LIN {X 0,Y 298.466,Z 479.305,A -85,B 0,C 180,E1 -16236.813,E2 -16236.813} C_VEL
LIN {X 0,Y 298.452,Z 479.311,A -85,B 0,C 180,E1 -16241.25,E2 -16241.25} C_VEL
LIN {X 0,Y 298.537,Z 479.479,A -85,B 0,C 180,E1 -16243.984,E2 -16243.984} C_VEL
LIN {X 0,Y 299.451,Z 484.848,A -85,B 0,C 180,E1 -16247.917,E2 -16247.917} C_VEL
LIN {X 0,Y 300.419,Z 490.228,A -85,B 0,C 180,E1 -16251.688,E2 -16251.688} C_VEL
LIN {X 0,Y 300.571,Z 494.055,A -85,B 0,C 180,E1 -16254.229,E2 -16254.229} C_VEL
LIN {X 0,Y 299.738,Z 499.296,A -85,B 0,C 180,E1 -16257.575,E2 -16257.575} C_VEL
LIN {X 0,Y 298.893,Z 505.042,A -85,B 0,C 180,E1 -16261.182,E2 -16261.182} C_VEL
LIN {X 0,Y 297.961,Z 512.224,A -85,B 0,C 180,E1 -16265.621,E2 -16265.621} C_VEL
LIN {X 0,Y 297.495,Z 517.191,A -85,B 0,C 180,E1 -16268.634,E2 -16268.634} C_VEL
LIN {X 0,Y 298.743,Z 530.872,A -85,B 0,C 180,E1 -16269.444,E2 -16269.444} C_VEL
LIN {X 0,Y 300.095,Z 544.162,A -85,B 0,C 180,E1 -16270.512,E2 -16270.512} C_VEL
LIN {X 0,Y 301.357,Z 557.073,A -85,B 0,C 180,E1 -16271.825,E2 -16271.825} C_VEL
LIN {X 0,Y 301.113,Z 562.88,A -85,B 0,C 180,E1 -16272.512,E2 -16272.512} C_VEL
LIN {X 0,Y 299.918,Z 574.212,A -85,B 0,C 180,E1 -16274.077,E2 -16274.077} C_VEL
LIN {X 0,Y 298.966,Z 583.854,A -85,B 0,C 180,E1 -16275.71,E2 -16275.71} C_VEL
LIN {X 0,Y 298.052,Z 593.552,A -85,B 0,C 180,E1 -16277.748,E2 -16277.748} C_VEL
LIN {X 0,Y 297.384,Z 601.387,A -85,B 0,C 180,E1 -16279.791,E2 -16279.791} C_VEL
LIN {X 0,Y 297.034,Z 607.671,A -85,B 0,C 180,E1 -16281.839,E2 -16281.839} C_VEL
LIN {X 0,Y 296.864,Z 612.635,A -85,B 0,C 180,E1 -16283.887,E2 -16283.887} C_VEL
LIN {X 0,Y 296.808,Z 616.412,A -85,B 0,C 180,E1 -16285.927,E2 -16285.927} C_VEL
LIN {X 0,Y 296.812,Z 618.317,A -85,B 0,C 180,E1 -16287.286,E2 -16287.286} C_VEL
LIN {X 0,Y 296.996,Z 619.803,A -85,B 0,C 180,E1 -16288.644,E2 -16288.644} C_VEL
LIN {X 0,Y 296.994,Z 620.81,A -85,B 0,C 180,E1 -16290,E2 -16290} C_VEL
LIN {X 0,Y 296.862,Z 621.357,A -85,B 0,C 180,E1 -16291.357,E2 -16291.357} C_VEL
LIN {X 0,Y 296.64,Z 621.229,A -85,B 0,C 180,E1 -16294.076,E2 -16294.076} C_VEL
LIN {X 0,Y 296.595,Z 620.43,A -85,B 0,C 180,E1 -16295.607,E2 -16295.607} C_VEL
LIN {X 0,Y 296.89,Z 617.954,A -85,B 0,C 180,E1 -16298.166,E2 -16298.166} C_VEL
LIN {X 0,Y 297.683,Z 613.764,A -85,B 0,C 180,E1 -16300.887,E2 -16300.887} C_VEL
LIN {X 0,Y 298.649,Z 609.478,A -85,B 0,C 180,E1 -16302.919,E2 -16302.919} C_VEL
LIN {X 0,Y 300.437,Z 603.094,A -85,B 0,C 180,E1 -16305.258,E2 -16305.258} C_VEL
LIN {X 0,Y 302.414,Z 595.236,A -85,B 0,C 180,E1 -16307.585,E2 -16307.585} C_VEL
LIN {X 0,Y 304.966,Z 586.959,A -85,B 0,C 180,E1 -16309.522,E2 -16309.522} C_VEL
LIN {X 0,Y 307.811,Z 577.052,A -85,B 0,C 180,E1 -16311.427,E2 -16311.427} C_VEL
LIN {X 0,Y 309.967,Z 569.372,A -85,B 0,C 180,E1 -16312.672,E2 -16312.672} C_VEL
LIN {X 0,Y 311.299,Z 559.086,A -85,B 0,C 180,E1 -16314.278,E2 -16314.278} C_VEL
LIN {X 0,Y 311.377,Z 550.475,A -85,B 0,C 180,E1 -16315.638,E2 -16315.638} C_VEL
LIN {X 0,Y 310.206,Z 538.996,A -85,B 0,C 180,E1 -16317.496,E2 -16317.496} C_VEL
LIN {X 0,Y 307.841,Z 527.667,A -85,B 0,C 180,E1 -16319.496,E2 -16319.496} C_VEL
LIN {X 0,Y 305.431,Z 518.991,A -85,B 0,C 180,E1 -16321.194,E2 -16321.194} C_VEL
LIN {X 0,Y 303.143,Z 512.4,A -85,B 0,C 180,E1 -16322.676,E2 -16322.676} C_VEL
LIN {X 0,Y 301.622,Z 508.711,A -85,B 0,C 180,E1 -16323.642,E2 -16323.642} C_VEL
LIN {X 0,Y 301.271,Z 506.687,A -85,B 0,C 180,E1 -16324.047,E2 -16324.047} C_VEL
LIN {X 0,Y 302.094,Z 503.342,A -85,B 0,C 180,E1 -16327.22,E2 -16327.22} C_VEL
LIN {X 0,Y 302.148,Z 501.053,A -85,B 0,C 180,E1 -16329.863,E2 -16329.863} C_VEL
LIN {X 0,Y 301.802,Z 498.422,A -85,B 0,C 180,E1 -16333.789,E2 -16333.789} C_VEL
LIN {X 0,Y 301.46,Z 496.683,A -85,B 0,C 180,E1 -16337.462,E2 -16337.462} C_VEL
LIN {X 0,Y 301.194,Z 495.638,A -85,B 0,C 180,E1 -16340.949,E2 -16340.949} C_VEL
LIN {X 0,Y 300.84,Z 495.191,A -85,B 0,C 180,E1 -16344.266,E2 -16344.266} C_VEL
LIN {X 0,Y 300.63,Z 495.276,A -85,B 0,C 180,E1 -16345.923,E2 -16345.923} C_VEL
LIN {X 0,Y 301.106,Z 496.736,A -85,B 0,C 180,E1 -16346.358,E2 -16346.358} C_VEL
LIN {X 0,Y 301.952,Z 498.177,A -85,B 0,C 180,E1 -16346.921,E2 -16346.921} C_VEL
LIN {X 0,Y 303.759,Z 499.965,A -85,B 0,C 180,E1 -16347.85,E2 -16347.85} C_VEL
LIN {X 0,Y 304.765,Z 502.419,A -85,B 0,C 180,E1 -16348.566,E2 -16348.566} C_VEL
LIN {X 0,Y 306.416,Z 504.69,A -85,B 0,C 180,E1 -16349.405,E2 -16349.405} C_VEL
LIN {X 0,Y 306.908,Z 506.071,A -85,B 0,C 180,E1 -16349.749,E2 -16349.749} C_VEL
LIN {X 0,Y 308.354,Z 508.316,A -85,B 0,C 180,E1 -16350.508,E2 -16350.508} C_VEL
LIN {X 0,Y 312.476,Z 517.896,A -85,B 0,C 180,E1 -16352.944,E2 -16352.944} C_VEL
LIN {X 0,Y 315.184,Z 526.862,A -85,B 0,C 180,E1 -16354.934,E2 -16354.934} C_VEL
LIN {X 0,Y 316.223,Z 532.587,A -85,B 0,C 180,E1 -16356.098,E2 -16356.098} C_VEL
LIN {X 0,Y 312.862,Z 544.975,A -85,B 0,C 180,E1 -16357.898,E2 -16357.898} C_VEL
LIN {X 0,Y 309.781,Z 555.156,A -85,B 0,C 180,E1 -16359.759,E2 -16359.759} C_VEL
LIN {X 0,Y 306.983,Z 563.531,A -85,B 0,C 180,E1 -16361.652,E2 -16361.652} C_VEL
LIN {X 0,Y 304.706,Z 570.437,A -85,B 0,C 180,E1 -16363.588,E2 -16363.588} C_VEL
LIN {X 0,Y 302.42,Z 576.841,A -85,B 0,C 180,E1 -16365.877,E2 -16365.877} C_VEL
LIN {X 0,Y 300.729,Z 581.193,A -85,B 0,C 180,E1 -16367.859,E2 -16367.859} C_VEL
LIN {X 0,Y 299.962,Z 583.522,A -85,B 0,C 180,E1 -16369.197,E2 -16369.197} C_VEL
LIN {X 0,Y 299.12,Z 585.612,A -85,B 0,C 180,E1 -16370.687,E2 -16370.687} C_VEL
LIN {X 0,Y 297.885,Z 588.001,A -85,B 0,C 180,E1 -16373.226,E2 -16373.226} C_VEL
LIN {X 0,Y 297.69,Z 588.691,A -85,B 0,C 180,E1 -16374.582,E2 -16374.582} C_VEL
LIN {X 0,Y 297.438,Z 589,A -85,B 0,C 180,E1 -16375.935,E2 -16375.935} C_VEL
LIN {X 0,Y 296.934,Z 588.398,A -85,B 0,C 180,E1 -16378.644,E2 -16378.644} C_VEL
LIN {X 0,Y 296.812,Z 587.512,A -85,B 0,C 180,E1 -16380,E2 -16380} C_VEL
LIN {X 0,Y 296.762,Z 586.21,A -85,B 0,C 180,E1 -16381.357,E2 -16381.357} C_VEL
LIN {X 0,Y 296.845,Z 583.461,A -85,B 0,C 180,E1 -16383.394,E2 -16383.394} C_VEL
LIN {X 0,Y 297.012,Z 579.68,A -85,B 0,C 180,E1 -16385.432,E2 -16385.432} C_VEL
LIN {X 0,Y 297.346,Z 574.78,A -85,B 0,C 180,E1 -16387.47,E2 -16387.47} C_VEL
LIN {X 0,Y 297.88,Z 567.471,A -85,B 0,C 180,E1 -16389.849,E2 -16389.849} C_VEL
LIN {X 0,Y 298.614,Z 559.653,A -85,B 0,C 180,E1 -16391.885,E2 -16391.885} C_VEL
LIN {X 0,Y 299.575,Z 549.967,A -85,B 0,C 180,E1 -16393.914,E2 -16393.914} C_VEL
LIN {X 0,Y 300.544,Z 540.158,A -85,B 0,C 180,E1 -16395.6,E2 -16395.6} C_VEL
LIN {X 0,Y 301.436,Z 530.908,A -85,B 0,C 180,E1 -16396.92,E2 -16396.92} C_VEL
LIN {X 0,Y 302.482,Z 519.263,A -85,B 0,C 180,E1 -16398.281,E2 -16398.281} C_VEL
LIN {X 0,Y 302.839,Z 514.221,A -85,B 0,C 180,E1 -16398.784,E2 -16398.784} C_VEL
LIN {X 0,Y 300.737,Z 502.562,A -85,B 0,C 180,E1 -16399.877,E2 -16399.877} C_VEL
LIN {X 0,Y 298.12,Z 489.054,A -85,B 0,C 180,E1 -16400.877,E2 -16400.877} C_VEL
LIN {X 0,Y 297.077,Z 483.361,A -85,B 0,C 180,E1 -16401.239,E2 -16401.239} C_VEL
LIN {X 0,Y 297.196,Z 479.837,A -85,B 0,C 180,E1 -16405.193,E2 -16405.193} C_VEL
LIN {X 0,Y 297.331,Z 479.45,A -85,B 0,C 180,E1 -16406.687,E2 -16406.687} C_VEL
LIN {X 0,Y 297.686,Z 479.402,A -85,B 0,C 180,E1 -16409.722,E2 -16409.722} C_VEL
LIN {X 0,Y 297.986,Z 479.364,A -85,B 0,C 180,E1 -16412.852,E2 -16412.852} C_VEL
LIN {X 0,Y 298.373,Z 479.317,A -85,B 0,C 180,E1 -16416.788,E2 -16416.788} C_VEL
LIN {X 0,Y 298.399,Z 479.312,A -85,B 0,C 180,E1 -16419.488,E2 -16419.488} C_VEL
LIN {X 0,Y 298.402,Z 479.311,A -85,B 0,C 180,E1 -16423.103,E2 -16423.103} C_VEL
LIN {X 0,Y 298.407,Z 479.312,A -85,B 0,C 180,E1 -16426.921,E2 -16426.921} C_VEL
LIN {X 0,Y 298.419,Z 479.309,A -85,B 0,C 180,E1 -16431.004,E2 -16431.004} C_VEL
LIN {X 0,Y 298.425,Z 479.312,A -85,B 0,C 180,E1 -16433.931,E2 -16433.931} C_VEL
LIN {X 0,Y 298.399,Z 479.316,A -85,B 0,C 180,E1 -16437.984,E2 -16437.984} C_VEL
LIN {X 0,Y 298.463,Z 479.307,A -85,B 0,C 180,E1 -16441.904,E2 -16441.904} C_VEL
LIN {X 0,Y 298.49,Z 479.301,A -85,B 0,C 180,E1 -16444.924,E2 -16444.924} C_VEL
LIN {X 0,Y 298.455,Z 479.305,A -85,B 0,C 180,E1 -16449.315,E2 -16449.315} C_VEL
LIN {X 0,Y 298.543,Z 479.299,A -85,B 0,C 180,E1 -16452.179,E2 -16452.179} C_VEL
LIN {X 0,Y 298.598,Z 479.287,A -85,B 0,C 180,E1 -16454.995,E2 -16454.995} C_VEL
LIN {X 0,Y 298.597,Z 479.287,A -85,B 0,C 180,E1 -16459.146,E2 -16459.146} C_VEL
LIN {X 0,Y 298.745,Z 479.273,A -85,B 0,C 180,E1 -16461.885,E2 -16461.885} C_VEL
LIN {X 0,Y 298.661,Z 479.28,A -85,B 0,C 180,E1 -16464.599,E2 -16464.599} C_VEL
LIN {X 0,Y 298.927,Z 479.247,A -85,B 0,C 180,E1 -16468.653,E2 -16468.653} C_VEL
LIN {X 0,Y 298.929,Z 479.247,A -85,B 0,C 180,E1 -16471.347,E2 -16471.347} C_VEL
LIN {X 0,Y 298.649,Z 479.281,A -85,B 0,C 180,E1 -16475.401,E2 -16475.401} C_VEL
LIN {X 0,Y 298.718,Z 479.276,A -85,B 0,C 180,E1 -16478.115,E2 -16478.115} C_VEL
LIN {X 0,Y 298.558,Z 479.294,A -85,B 0,C 180,E1 -16482.231,E2 -16482.231} C_VEL
LIN {X 0,Y 298.61,Z 479.286,A -85,B 0,C 180,E1 -16485.209,E2 -16485.209} C_VEL
LIN {X 0,Y 298.544,Z 479.295,A -85,B 0,C 180,E1 -16489.243,E2 -16489.243} C_VEL
LIN {X 0,Y 298.461,Z 479.307,A -85,B 0,C 180,E1 -16493.597,E2 -16493.597} C_VEL
LIN {X 0,Y 298.49,Z 479.301,A -85,B 0,C 180,E1 -16496.574,E2 -16496.574} C_VEL
LIN {X 0,Y 298.419,Z 479.313,A -85,B 0,C 180,E1 -16499.641,E2 -16499.641} C_VEL
LIN {X 0,Y 298.398,Z 479.312,A -85,B 0,C 180,E1 -16502.8,E2 -16502.8} C_VEL
LIN {X 0,Y 298.467,Z 479.303,A -85,B 0,C 180,E1 -16506.812,E2 -16506.812} C_VEL
LIN {X 0,Y 298.389,Z 479.313,A -85,B 0,C 180,E1 -16511.087,E2 -16511.087} C_VEL
LIN {X 0,Y 298.4,Z 479.313,A -85,B 0,C 180,E1 -16513.103,E2 -16513.103} C_VEL
LIN {X 0,Y 298.404,Z 479.311,A -85,B 0,C 180,E1 -16516.92,E2 -16516.92} C_VEL
LIN {X 0,Y 298.416,Z 479.31,A -85,B 0,C 180,E1 -16521.003,E2 -16521.003} C_VEL
LIN {X 0,Y 298.42,Z 479.313,A -85,B 0,C 180,E1 -16523.93,E2 -16523.93} C_VEL
LIN {X 0,Y 298.397,Z 479.315,A -85,B 0,C 180,E1 -16527.983,E2 -16527.983} C_VEL
LIN {X 0,Y 298.465,Z 479.307,A -85,B 0,C 180,E1 -16531.904,E2 -16531.904} C_VEL
LIN {X 0,Y 298.487,Z 479.301,A -85,B 0,C 180,E1 -16534.924,E2 -16534.924} C_VEL
LIN {X 0,Y 298.451,Z 479.308,A -85,B 0,C 180,E1 -16539.315,E2 -16539.315} C_VEL
LIN {X 0,Y 298.539,Z 479.295,A -85,B 0,C 180,E1 -16542.179,E2 -16542.179} C_VEL
LIN {X 0,Y 298.594,Z 479.288,A -85,B 0,C 180,E1 -16544.994,E2 -16544.994} C_VEL
LIN {X 0,Y 298.595,Z 479.29,A -85,B 0,C 180,E1 -16549.146,E2 -16549.146} C_VEL
LIN {X 0,Y 298.759,Z 479.269,A -85,B 0,C 180,E1 -16551.886,E2 -16551.886} C_VEL
LIN {X 0,Y 298.661,Z 479.279,A -85,B 0,C 180,E1 -16554.599,E2 -16554.599} C_VEL
LIN {X 0,Y 298.925,Z 479.247,A -85,B 0,C 180,E1 -16558.652,E2 -16558.652} C_VEL
LIN {X 0,Y 298.924,Z 479.25,A -85,B 0,C 180,E1 -16561.347,E2 -16561.347} C_VEL
LIN {X 0,Y 298.618,Z 479.284,A -85,B 0,C 180,E1 -16563.886,E2 -16563.886} C_VEL
LIN {X 0,Y 297.887,Z 479.382,A -85,B 0,C 180,E1 -16565.012,E2 -16565.012} C_VEL
LIN {X 0,Y 295.114,Z 479.733,A -85,B 0,C 180,E1 -16566.85,E2 -16566.85} C_VEL
LIN {X 0,Y 291.972,Z 480.118,A -85,B 0,C 180,E1 -16569.104,E2 -16569.104} C_VEL
LIN {X 0,Y 291.609,Z 480.159,A -85,B 0,C 180,E1 -16569.881,E2 -16569.881} C_VEL
LIN {X 0,Y 291.522,Z 480.17,A -85,B 0,C 180,E1 -16573.95,E2 -16573.95} C_VEL
LIN {X 0,Y 291.487,Z 480.174,A -85,B 0,C 180,E1 -16576.818,E2 -16576.818} C_VEL
LIN {X 0,Y 291.45,Z 480.178,A -85,B 0,C 180,E1 -16579.875,E2 -16579.875} C_VEL
LIN {X 0,Y 291.399,Z 480.184,A -85,B 0,C 180,E1 -16584.205,E2 -16584.205} C_VEL
LIN {X 0,Y 291.418,Z 480.186,A -85,B 0,C 180,E1 -16587.272,E2 -16587.272} C_VEL
LIN {X 0,Y 291.334,Z 480.192,A -85,B 0,C 180,E1 -16590.437,E2 -16590.437} C_VEL
LIN {X 0,Y 291.344,Z 480.193,A -85,B 0,C 180,E1 -16593.698,E2 -16593.698} C_VEL
LIN {X 0,Y 291.399,Z 480.188,A -85,B 0,C 180,E1 -16597.26,E2 -16597.26} C_VEL
LIN {X 0,Y 291.4,Z 480.185,A -85,B 0,C 180,E1 -16600.631,E2 -16600.631} C_VEL
LIN {X 0,Y 291.489,Z 480.238,A -85,B 0,C 180,E1 -16603.748,E2 -16603.748} C_VEL
LIN {X 0,Y 292.493,Z 486.094,A -85,B 0,C 180,E1 -16608.147,E2 -16608.147} C_VEL
LIN {X 0,Y 293.31,Z 490.731,A -85,B 0,C 180,E1 -16611.466,E2 -16611.466} C_VEL
LIN {X 0,Y 293.549,Z 493.289,A -85,B 0,C 180,E1 -16613.235,E2 -16613.235} C_VEL
LIN {X 0,Y 293.16,Z 497.014,A -85,B 0,C 180,E1 -16615.711,E2 -16615.711} C_VEL
LIN {X 0,Y 292.082,Z 503.661,A -85,B 0,C 180,E1 -16620.023,E2 -16620.023} C_VEL
LIN {X 0,Y 291.131,Z 510.266,A -85,B 0,C 180,E1 -16624.245,E2 -16624.245} C_VEL
LIN {X 0,Y 290.418,Z 517.025,A -85,B 0,C 180,E1 -16628.39,E2 -16628.39} C_VEL
LIN {X 0,Y 291.665,Z 530.669,A -85,B 0,C 180,E1 -16629.225,E2 -16629.225} C_VEL
LIN {X 0,Y 293.019,Z 544.552,A -85,B 0,C 180,E1 -16630.38,E2 -16630.38} C_VEL
LIN {X 0,Y 294.281,Z 557.344,A -85,B 0,C 180,E1 -16631.733,E2 -16631.733} C_VEL
LIN {X 0,Y 293.898,Z 564.374,A -85,B 0,C 180,E1 -16632.608,E2 -16632.608} C_VEL
LIN {X 0,Y 292.718,Z 575.145,A -85,B 0,C 180,E1 -16634.181,E2 -16634.181} C_VEL
LIN {X 0,Y 291.697,Z 585.479,A -85,B 0,C 180,E1 -16636.059,E2 -16636.059} C_VEL
LIN {X 0,Y 290.819,Z 594.796,A -85,B 0,C 180,E1 -16638.147,E2 -16638.147} C_VEL
LIN {X 0,Y 290.249,Z 602.267,A -85,B 0,C 180,E1 -16640.242,E2 -16640.242} C_VEL
LIN {X 0,Y 289.929,Z 608.278,A -85,B 0,C 180,E1 -16642.339,E2 -16642.339} C_VEL
LIN {X 0,Y 289.863,Z 613.015,A -85,B 0,C 180,E1 -16644.435,E2 -16644.435} C_VEL
LIN {X 0,Y 289.753,Z 615.522,A -85,B 0,C 180,E1 -16645.827,E2 -16645.827} C_VEL
LIN {X 0,Y 289.74,Z 617.505,A -85,B 0,C 180,E1 -16647.22,E2 -16647.22} C_VEL
LIN {X 0,Y 289.938,Z 619.053,A -85,B 0,C 180,E1 -16648.611,E2 -16648.611} C_VEL
LIN {X 0,Y 289.939,Z 620.147,A -85,B 0,C 180,E1 -16650,E2 -16650} C_VEL
LIN {X 0,Y 289.773,Z 620.789,A -85,B 0,C 180,E1 -16651.39,E2 -16651.39} C_VEL
LIN {X 0,Y 289.551,Z 620.801,A -85,B 0,C 180,E1 -16654.176,E2 -16654.176} C_VEL
LIN {X 0,Y 289.602,Z 619.229,A -85,B 0,C 180,E1 -16656.97,E2 -16656.97} C_VEL
LIN {X 0,Y 290.21,Z 616.025,A -85,B 0,C 180,E1 -16659.76,E2 -16659.76} C_VEL
LIN {X 0,Y 291.286,Z 611.2,A -85,B 0,C 180,E1 -16662.542,E2 -16662.542} C_VEL
LIN {X 0,Y 292.75,Z 606.428,A -85,B 0,C 180,E1 -16664.6,E2 -16664.6} C_VEL
LIN {X 0,Y 294.73,Z 599.496,A -85,B 0,C 180,E1 -16666.985,E2 -16666.985} C_VEL
LIN {X 0,Y 297.014,Z 592.228,A -85,B 0,C 180,E1 -16668.987,E2 -16668.987} C_VEL
LIN {X 0,Y 299.844,Z 583.583,A -85,B 0,C 180,E1 -16670.944,E2 -16670.944} C_VEL
LIN {X 0,Y 302.506,Z 575.043,A -85,B 0,C 180,E1 -16672.541,E2 -16672.541} C_VEL
LIN {X 0,Y 304.015,Z 569.384,A -85,B 0,C 180,E1 -16673.502,E2 -16673.502} C_VEL
LIN {X 0,Y 305.303,Z 561.033,A -85,B 0,C 180,E1 -16674.885,E2 -16674.885} C_VEL
LIN {X 0,Y 305.532,Z 551.878,A -85,B 0,C 180,E1 -16676.418,E2 -16676.418} C_VEL
LIN {X 0,Y 304.602,Z 541.064,A -85,B 0,C 180,E1 -16678.31,E2 -16678.31} C_VEL
LIN {X 0,Y 302.739,Z 531.064,A -85,B 0,C 180,E1 -16680.23,E2 -16680.23} C_VEL
LIN {X 0,Y 300.864,Z 523.19,A -85,B 0,C 180,E1 -16681.895,E2 -16681.895} C_VEL
LIN {X 0,Y 299.552,Z 518.592,A -85,B 0,C 180,E1 -16682.969,E2 -16682.969} C_VEL
LIN {X 0,Y 297.801,Z 513.56,A -85,B 0,C 180,E1 -16684.311,E2 -16684.311} C_VEL
LIN {X 0,Y 297.659,Z 512.608,A -85,B 0,C 180,E1 -16684.518,E2 -16684.518} C_VEL
LIN {X 0,Y 295.612,Z 508.107,A -85,B 0,C 180,E1 -16686.067,E2 -16686.067} C_VEL
LIN {X 0,Y 295.034,Z 505.141,A -85,B 0,C 180,E1 -16686.918,E2 -16686.918} C_VEL
LIN {X 0,Y 295.199,Z 503.926,A -85,B 0,C 180,E1 -16688.244,E2 -16688.244} C_VEL
LIN {X 0,Y 295.16,Z 502.235,A -85,B 0,C 180,E1 -16690.364,E2 -16690.364} C_VEL
LIN {X 0,Y 294.894,Z 500.053,A -85,B 0,C 180,E1 -16693.721,E2 -16693.721} C_VEL
LIN {X 0,Y 294.53,Z 498.2,A -85,B 0,C 180,E1 -16697.708,E2 -16697.708} C_VEL
LIN {X 0,Y 294.354,Z 497.513,A -85,B 0,C 180,E1 -16699.86,E2 -16699.86} C_VEL
LIN {X 0,Y 294.116,Z 497.014,A -85,B 0,C 180,E1 -16702.839,E2 -16702.839} C_VEL
LIN {X 0,Y 295.223,Z 499.509,A -85,B 0,C 180,E1 -16704.038,E2 -16704.038} C_VEL
LIN {X 0,Y 297.165,Z 501.335,A -85,B 0,C 180,E1 -16705.417,E2 -16705.417} C_VEL
LIN {X 0,Y 298.652,Z 504.229,A -85,B 0,C 180,E1 -16706.606,E2 -16706.606} C_VEL
LIN {X 0,Y 300.119,Z 505.816,A -85,B 0,C 180,E1 -16707.462,E2 -16707.462} C_VEL
LIN {X 0,Y 301.121,Z 508.24,A -85,B 0,C 180,E1 -16708.239,E2 -16708.239} C_VEL
LIN {X 0,Y 301.971,Z 509.364,A -85,B 0,C 180,E1 -16708.742,E2 -16708.742} C_VEL
LIN {X 0,Y 304.883,Z 515.521,A -85,B 0,C 180,E1 -16710.662,E2 -16710.662} C_VEL
LIN {X 0,Y 308.306,Z 524.86,A -85,B 0,C 180,E1 -16713.119,E2 -16713.119} C_VEL
LIN {X 0,Y 310.177,Z 532.971,A -85,B 0,C 180,E1 -16715.003,E2 -16715.003} C_VEL
LIN {X 0,Y 310.364,Z 534.297,A -85,B 0,C 180,E1 -16715.289,E2 -16715.289} C_VEL
LIN {X 0,Y 309.843,Z 537.437,A -85,B 0,C 180,E1 -16715.785,E2 -16715.785} C_VEL
LIN {X 0,Y 306.669,Z 547.839,A -85,B 0,C 180,E1 -16717.427,E2 -16717.427} C_VEL
LIN {X 0,Y 303.434,Z 557.555,A -85,B 0,C 180,E1 -16719.316,E2 -16719.316} C_VEL
LIN {X 0,Y 300.51,Z 565.566,A -85,B 0,C 180,E1 -16721.242,E2 -16721.242} C_VEL
LIN {X 0,Y 297.689,Z 573.08,A -85,B 0,C 180,E1 -16723.543,E2 -16723.543} C_VEL
LIN {X 0,Y 295.7,Z 578.283,A -85,B 0,C 180,E1 -16725.549,E2 -16725.549} C_VEL
LIN {X 0,Y 293.904,Z 582.416,A -85,B 0,C 180,E1 -16727.572,E2 -16727.572} C_VEL
LIN {X 0,Y 293.078,Z 584.589,A -85,B 0,C 180,E1 -16728.94,E2 -16728.94} C_VEL
LIN {X 0,Y 291.473,Z 587.758,A -85,B 0,C 180,E1 -16731.682,E2 -16731.682} C_VEL
LIN {X 0,Y 290.873,Z 588.76,A -85,B 0,C 180,E1 -16733.062,E2 -16733.062} C_VEL
LIN {X 0,Y 290.635,Z 589.327,A -85,B 0,C 180,E1 -16734.45,E2 -16734.45} C_VEL
LIN {X 0,Y 290.369,Z 589.505,A -85,B 0,C 180,E1 -16735.836,E2 -16735.836} C_VEL
LIN {X 0,Y 289.845,Z 588.74,A -85,B 0,C 180,E1 -16738.611,E2 -16738.611} C_VEL
LIN {X 0,Y 289.717,Z 587.746,A -85,B 0,C 180,E1 -16740,E2 -16740} C_VEL
LIN {X 0,Y 289.673,Z 586.323,A -85,B 0,C 180,E1 -16741.391,E2 -16741.391} C_VEL
LIN {X 0,Y 289.777,Z 583.417,A -85,B 0,C 180,E1 -16743.476,E2 -16743.476} C_VEL
LIN {X 0,Y 289.947,Z 578.622,A -85,B 0,C 180,E1 -16745.965,E2 -16745.965} C_VEL
LIN {X 0,Y 290.396,Z 572.51,A -85,B 0,C 180,E1 -16748.35,E2 -16748.35} C_VEL
LIN {X 0,Y 291.071,Z 564.428,A -85,B 0,C 180,E1 -16750.786,E2 -16750.786} C_VEL
LIN {X 0,Y 291.897,Z 555.777,A -85,B 0,C 180,E1 -16752.869,E2 -16752.869} C_VEL
LIN {X 0,Y 293.033,Z 545.097,A -85,B 0,C 180,E1 -16754.941,E2 -16754.941} C_VEL
LIN {X 0,Y 294.202,Z 534.097,A -85,B 0,C 180,E1 -16756.659,E2 -16756.659} C_VEL
LIN {X 0,Y 295.258,Z 521.873,A -85,B 0,C 180,E1 -16758.205,E2 -16758.205} C_VEL
LIN {X 0,Y 295.753,Z 515.364,A -85,B 0,C 180,E1 -16758.892,E2 -16758.892} C_VEL
LIN {X 0,Y 294.403,Z 506.887,A -85,B 0,C 180,E1 -16759.734,E2 -16759.734} C_VEL
LIN {X 0,Y 292.017,Z 494.407,A -85,B 0,C 180,E1 -16760.767,E2 -16760.767} C_VEL
LIN {X 0,Y 290.011,Z 483.742,A -85,B 0,C 180,E1 -16761.502,E2 -16761.502} C_VEL
LIN {X 0,Y 290.054,Z 481.255,A -85,B 0,C 180,E1 -16764.325,E2 -16764.325} C_VEL
LIN {X 0,Y 290.218,Z 480.336,A -85,B 0,C 180,E1 -16765.843,E2 -16765.843} C_VEL
LIN {X 0,Y 290.616,Z 480.282,A -85,B 0,C 180,E1 -16769.472,E2 -16769.472} C_VEL
LIN {X 0,Y 290.907,Z 480.25,A -85,B 0,C 180,E1 -16772.267,E2 -16772.267} C_VEL
LIN {X 0,Y 291.182,Z 480.211,A -85,B 0,C 180,E1 -16775.4,E2 -16775.4} C_VEL
LIN {X 0,Y 291.319,Z 480.194,A -85,B 0,C 180,E1 -16777.239,E2 -16777.239} C_VEL
LIN {X 0,Y 291.335,Z 480.193,A -85,B 0,C 180,E1 -16780.643,E2 -16780.643} C_VEL
LIN {X 0,Y 291.294,Z 480.201,A -85,B 0,C 180,E1 -16784.402,E2 -16784.402} C_VEL
LIN {X 0,Y 291.33,Z 480.196,A -85,B 0,C 180,E1 -16788.404,E2 -16788.404} C_VEL
LIN {X 0,Y 291.368,Z 480.187,A -85,B 0,C 180,E1 -16791.16,E2 -16791.16} C_VEL
LIN {X 0,Y 291.366,Z 480.19,A -85,B 0,C 180,E1 -16794.626,E2 -16794.626} C_VEL
LIN {X 0,Y 291.376,Z 480.19,A -85,B 0,C 180,E1 -16797.951,E2 -16797.951} C_VEL
LIN {X 0,Y 291.382,Z 480.186,A -85,B 0,C 180,E1 -16801.158,E2 -16801.158} C_VEL
LIN {X 0,Y 291.419,Z 480.186,A -85,B 0,C 180,E1 -16804.272,E2 -16804.272} C_VEL
LIN {X 0,Y 291.387,Z 480.185,A -85,B 0,C 180,E1 -16807.3,E2 -16807.3} C_VEL
LIN {X 0,Y 291.463,Z 480.18,A -85,B 0,C 180,E1 -16810.27,E2 -16810.27} C_VEL
LIN {X 0,Y 291.56,Z 480.165,A -85,B 0,C 180,E1 -16814.624,E2 -16814.624} C_VEL
LIN {X 0,Y 291.54,Z 480.166,A -85,B 0,C 180,E1 -16818.88,E2 -16818.88} C_VEL
LIN {X 0,Y 291.692,Z 480.15,A -85,B 0,C 180,E1 -16821.688,E2 -16821.688} C_VEL
LIN {X 0,Y 291.631,Z 480.156,A -85,B 0,C 180,E1 -16824.468,E2 -16824.468} C_VEL
LIN {X 0,Y 291.893,Z 480.123,A -85,B 0,C 180,E1 -16828.62,E2 -16828.62} C_VEL
LIN {X 0,Y 291.895,Z 480.123,A -85,B 0,C 180,E1 -16831.379,E2 -16831.379} C_VEL
LIN {X 0,Y 291.617,Z 480.158,A -85,B 0,C 180,E1 -16835.532,E2 -16835.532} C_VEL
LIN {X 0,Y 291.678,Z 480.149,A -85,B 0,C 180,E1 -16838.919,E2 -16838.919} C_VEL
LIN {X 0,Y 291.525,Z 480.168,A -85,B 0,C 180,E1 -16842.531,E2 -16842.531} C_VEL
LIN {X 0,Y 291.559,Z 480.165,A -85,B 0,C 180,E1 -16845.376,E2 -16845.376} C_VEL
LIN {X 0,Y 291.454,Z 480.182,A -85,B 0,C 180,E1 -16849.874,E2 -16849.874} C_VEL
LIN {X 0,Y 291.404,Z 480.186,A -85,B 0,C 180,E1 -16854.205,E2 -16854.205} C_VEL
LIN {X 0,Y 291.423,Z 480.182,A -85,B 0,C 180,E1 -16857.271,E2 -16857.271} C_VEL
LIN {X 0,Y 291.337,Z 480.192,A -85,B 0,C 180,E1 -16860.437,E2 -16860.437} C_VEL
LIN {X 0,Y 291.348,Z 480.195,A -85,B 0,C 180,E1 -16863.698,E2 -16863.698} C_VEL
LIN {X 0,Y 291.397,Z 480.185,A -85,B 0,C 180,E1 -16867.258,E2 -16867.258} C_VEL
LIN {X 0,Y 291.336,Z 480.191,A -85,B 0,C 180,E1 -16870.642,E2 -16870.642} C_VEL
LIN {X 0,Y 291.292,Z 480.198,A -85,B 0,C 180,E1 -16874.401,E2 -16874.401} C_VEL
LIN {X 0,Y 291.328,Z 480.193,A -85,B 0,C 180,E1 -16878.404,E2 -16878.404} C_VEL
LIN {X 0,Y 291.365,Z 480.189,A -85,B 0,C 180,E1 -16881.16,E2 -16881.16} C_VEL
LIN {X 0,Y 291.363,Z 480.189,A -85,B 0,C 180,E1 -16884.626,E2 -16884.626} C_VEL
LIN {X 0,Y 291.374,Z 480.19,A -85,B 0,C 180,E1 -16887.95,E2 -16887.95} C_VEL
LIN {X 0,Y 291.383,Z 480.187,A -85,B 0,C 180,E1 -16891.158,E2 -16891.158} C_VEL
LIN {X 0,Y 291.418,Z 480.182,A -85,B 0,C 180,E1 -16894.272,E2 -16894.272} C_VEL
LIN {X 0,Y 291.383,Z 480.188,A -85,B 0,C 180,E1 -16897.299,E2 -16897.299} C_VEL
LIN {X 0,Y 291.459,Z 480.177,A -85,B 0,C 180,E1 -16900.27,E2 -16900.27} C_VEL
LIN {X 0,Y 291.556,Z 480.163,A -85,B 0,C 180,E1 -16904.623,E2 -16904.623} C_VEL
LIN {X 0,Y 291.538,Z 480.167,A -85,B 0,C 180,E1 -16908.88,E2 -16908.88} C_VEL
LIN {X 0,Y 291.71,Z 480.149,A -85,B 0,C 180,E1 -16911.688,E2 -16911.688} C_VEL
LIN {X 0,Y 291.632,Z 480.155,A -85,B 0,C 180,E1 -16914.468,E2 -16914.468} C_VEL
LIN {X 0,Y 291.891,Z 480.123,A -85,B 0,C 180,E1 -16918.62,E2 -16918.62} C_VEL
LIN {X 0,Y 291.89,Z 480.127,A -85,B 0,C 180,E1 -16921.379,E2 -16921.379} C_VEL
LIN {X 0,Y 291.747,Z 480.142,A -85,B 0,C 180,E1 -16926.918,E2 -16926.918} C_VEL
LIN {X 0,Y 291.609,Z 480.159,A -85,B 0,C 180,E1 -16929.881,E2 -16929.881} C_VEL
LIN {X 0,Y 290.87,Z 480.253,A -85,B 0,C 180,E1 -16931.032,E2 -16931.032} C_VEL
LIN {X 0,Y 288.028,Z 480.605,A -85,B 0,C 180,E1 -16932.908,E2 -16932.908} C_VEL
LIN {X 0,Y 285.637,Z 480.906,A -85,B 0,C 180,E1 -16934.43,E2 -16934.43} C_VEL
LIN {X 0,Y 284.574,Z 481.038,A -85,B 0,C 180,E1 -16935.609,E2 -16935.609} C_VEL
LIN {X 0,Y 284.464,Z 481.049,A -85,B 0,C 180,E1 -16936.008,E2 -16936.008} C_VEL
LIN {X 0,Y 284.378,Z 481.058,A -85,B 0,C 180,E1 -16940.242,E2 -16940.242} C_VEL
LIN {X 0,Y 284.369,Z 481.061,A -85,B 0,C 180,E1 -16943.875,E2 -16943.875} C_VEL
LIN {X 0,Y 284.394,Z 481.06,A -85,B 0,C 180,E1 -16947.172,E2 -16947.172} C_VEL
LIN {X 0,Y 284.293,Z 481.074,A -85,B 0,C 180,E1 -16951.274,E2 -16951.274} C_VEL
LIN {X 0,Y 284.361,Z 481.065,A -85,B 0,C 180,E1 -16955.354,E2 -16955.354} C_VEL
LIN {X 0,Y 284.331,Z 481.064,A -85,B 0,C 180,E1 -16958.166,E2 -16958.166} C_VEL
LIN {X 0,Y 284.341,Z 481.064,A -85,B 0,C 180,E1 -16962.141,E2 -16962.141} C_VEL
LIN {X 0,Y 284.435,Z 481.169,A -85,B 0,C 180,E1 -16963.664,E2 -16963.664} C_VEL
LIN {X 0,Y 285.321,Z 486.329,A -85,B 0,C 180,E1 -16967.642,E2 -16967.642} C_VEL
LIN {X 0,Y 286.163,Z 490.991,A -85,B 0,C 180,E1 -16971.09,E2 -16971.09} C_VEL
LIN {X 0,Y 286.485,Z 493.758,A -85,B 0,C 180,E1 -16973.057,E2 -16973.057} C_VEL
LIN {X 0,Y 286.112,Z 497.472,A -85,B 0,C 180,E1 -16975.6,E2 -16975.6} C_VEL
LIN {X 0,Y 285.068,Z 503.522,A -85,B 0,C 180,E1 -16979.642,E2 -16979.642} C_VEL
LIN {X 0,Y 284.163,Z 509.476,A -85,B 0,C 180,E1 -16983.565,E2 -16983.565} C_VEL
LIN {X 0,Y 283.373,Z 516.221,A -85,B 0,C 180,E1 -16987.969,E2 -16987.969} C_VEL
LIN {X 0,Y 283.351,Z 516.442,A -85,B 0,C 180,E1 -16988.111,E2 -16988.111} C_VEL
LIN {X 0,Y 284.499,Z 530.072,A -85,B 0,C 180,E1 -16988.979,E2 -16988.979} C_VEL
LIN {X 0,Y 285.827,Z 543.775,A -85,B 0,C 180,E1 -16990.146,E2 -16990.146} C_VEL
LIN {X 0,Y 287.047,Z 555.823,A -85,B 0,C 180,E1 -16991.441,E2 -16991.441} C_VEL
LIN {X 0,Y 287.206,Z 560.398,A -85,B 0,C 180,E1 -16992.005,E2 -16992.005} C_VEL
LIN {X 0,Y 286.128,Z 570.715,A -85,B 0,C 180,E1 -16993.445,E2 -16993.445} C_VEL
LIN {X 0,Y 284.959,Z 581.786,A -85,B 0,C 180,E1 -16995.357,E2 -16995.357} C_VEL
LIN {X 0,Y 284.116,Z 590.214,A -85,B 0,C 180,E1 -16997.137,E2 -16997.137} C_VEL
LIN {X 0,Y 283.38,Z 598.489,A -85,B 0,C 180,E1 -16999.281,E2 -16999.281} C_VEL
LIN {X 0,Y 282.99,Z 605.171,A -85,B 0,C 180,E1 -17001.431,E2 -17001.431} C_VEL
LIN {X 0,Y 282.759,Z 611.01,A -85,B 0,C 180,E1 -17003.827,E2 -17003.827} C_VEL
LIN {X 0,Y 282.708,Z 614.529,A -85,B 0,C 180,E1 -17005.723,E2 -17005.723} C_VEL
LIN {X 0,Y 282.674,Z 616.637,A -85,B 0,C 180,E1 -17007.15,E2 -17007.15} C_VEL
LIN {X 0,Y 282.88,Z 618.264,A -85,B 0,C 180,E1 -17008.577,E2 -17008.577} C_VEL
LIN {X 0,Y 282.885,Z 619.433,A -85,B 0,C 180,E1 -17010,E2 -17010} C_VEL
LIN {X 0,Y 282.704,Z 620.169,A -85,B 0,C 180,E1 -17011.425,E2 -17011.425} C_VEL
LIN {X 0,Y 282.498,Z 620.489,A -85,B 0,C 180,E1 -17012.852,E2 -17012.852} C_VEL
LIN {X 0,Y 282.442,Z 619.945,A -85,B 0,C 180,E1 -17015.546,E2 -17015.546} C_VEL
LIN {X 0,Y 282.549,Z 618.968,A -85,B 0,C 180,E1 -17017.145,E2 -17017.145} C_VEL
LIN {X 0,Y 282.796,Z 617.688,A -85,B 0,C 180,E1 -17018.576,E2 -17018.576} C_VEL
LIN {X 0,Y 283.705,Z 613.887,A -85,B 0,C 180,E1 -17021.431,E2 -17021.431} C_VEL
LIN {X 0,Y 284.794,Z 609.99,A -85,B 0,C 180,E1 -17023.559,E2 -17023.559} C_VEL
LIN {X 0,Y 286.466,Z 605.074,A -85,B 0,C 180,E1 -17025.657,E2 -17025.657} C_VEL
LIN {X 0,Y 289.041,Z 596.908,A -85,B 0,C 180,E1 -17028.427,E2 -17028.427} C_VEL
LIN {X 0,Y 292.304,Z 587.856,A -85,B 0,C 180,E1 -17030.772,E2 -17030.772} C_VEL
LIN {X 0,Y 295.498,Z 578.584,A -85,B 0,C 180,E1 -17032.736,E2 -17032.736} C_VEL
LIN {X 0,Y 297.787,Z 571.41,A -85,B 0,C 180,E1 -17034.024,E2 -17034.024} C_VEL
LIN {X 0,Y 299.357,Z 562.824,A -85,B 0,C 180,E1 -17035.534,E2 -17035.534} C_VEL
LIN {X 0,Y 299.798,Z 553.604,A -85,B 0,C 180,E1 -17037.202,E2 -17037.202} C_VEL
LIN {X 0,Y 299.142,Z 543.021,A -85,B 0,C 180,E1 -17039.207,E2 -17039.207} C_VEL
LIN {X 0,Y 297.55,Z 532.97,A -85,B 0,C 180,E1 -17041.308,E2 -17041.308} C_VEL
LIN {X 0,Y 295.334,Z 523.352,A -85,B 0,C 180,E1 -17043.604,E2 -17043.604} C_VEL
LIN {X 0,Y 293.445,Z 516.85,A -85,B 0,C 180,E1 -17045.482,E2 -17045.482} C_VEL
LIN {X 0,Y 292.017,Z 512.479,A -85,B 0,C 180,E1 -17046.991,E2 -17046.991} C_VEL
LIN {X 0,Y 291.808,Z 511.164,A -85,B 0,C 180,E1 -17047.365,E2 -17047.365} C_VEL
LIN {X 0,Y 288.759,Z 504.955,A -85,B 0,C 180,E1 -17051.083,E2 -17051.083} C_VEL
LIN {X 0,Y 287.993,Z 501.758,A -85,B 0,C 180,E1 -17053.553,E2 -17053.553} C_VEL
LIN {X 0,Y 287.806,Z 500.62,A -85,B 0,C 180,E1 -17055.974,E2 -17055.974} C_VEL
LIN {X 0,Y 288.439,Z 501.626,A -85,B 0,C 180,E1 -17059.055,E2 -17059.055} C_VEL
LIN {X 0,Y 291.413,Z 503.822,A -85,B 0,C 180,E1 -17062.737,E2 -17062.737} C_VEL
LIN {X 0,Y 292.328,Z 505.915,A -85,B 0,C 180,E1 -17063.863,E2 -17063.863} C_VEL
LIN {X 0,Y 293.662,Z 507.266,A -85,B 0,C 180,E1 -17064.944,E2 -17064.944} C_VEL
LIN {X 0,Y 296.553,Z 512.134,A -85,B 0,C 180,E1 -17067.281,E2 -17067.281} C_VEL
LIN {X 0,Y 300.149,Z 519.879,A -85,B 0,C 180,E1 -17070.039,E2 -17070.039} C_VEL
LIN {X 0,Y 302.847,Z 527.89,A -85,B 0,C 180,E1 -17072.346,E2 -17072.346} C_VEL
LIN {X 0,Y 304.614,Z 536.548,A -85,B 0,C 180,E1 -17074.514,E2 -17074.514} C_VEL
LIN {X 0,Y 304.699,Z 537.826,A -85,B 0,C 180,E1 -17074.798,E2 -17074.798} C_VEL
LIN {X 0,Y 301.102,Z 549,A -85,B 0,C 180,E1 -17076.622,E2 -17076.622} C_VEL
LIN {X 0,Y 297.644,Z 558.575,A -85,B 0,C 180,E1 -17078.532,E2 -17078.532} C_VEL
LIN {X 0,Y 294.034,Z 567.576,A -85,B 0,C 180,E1 -17080.813,E2 -17080.813} C_VEL
LIN {X 0,Y 291.091,Z 574.794,A -85,B 0,C 180,E1 -17083.159,E2 -17083.159} C_VEL
LIN {X 0,Y 288.974,Z 579.689,A -85,B 0,C 180,E1 -17085.205,E2 -17085.205} C_VEL
LIN {X 0,Y 286.608,Z 584.705,A -85,B 0,C 180,E1 -17087.97,E2 -17087.97} C_VEL
LIN {X 0,Y 285.259,Z 587.491,A -85,B 0,C 180,E1 -17090.231,E2 -17090.231} C_VEL
LIN {X 0,Y 283.867,Z 589.466,A -85,B 0,C 180,E1 -17092.889,E2 -17092.889} C_VEL
LIN {X 0,Y 283.578,Z 589.924,A -85,B 0,C 180,E1 -17094.311,E2 -17094.311} C_VEL
LIN {X 0,Y 283.3,Z 590.016,A -85,B 0,C 180,E1 -17095.732,E2 -17095.732} C_VEL
LIN {X 0,Y 282.98,Z 589.737,A -85,B 0,C 180,E1 -17097.153,E2 -17097.153} C_VEL
LIN {X 0,Y 282.755,Z 589.038,A -85,B 0,C 180,E1 -17098.576,E2 -17098.576} C_VEL
LIN {X 0,Y 282.586,Z 586.427,A -85,B 0,C 180,E1 -17101.425,E2 -17101.425} C_VEL
LIN {X 0,Y 282.71,Z 583.358,A -85,B 0,C 180,E1 -17103.564,E2 -17103.564} C_VEL
LIN {X 0,Y 282.845,Z 579.26,A -85,B 0,C 180,E1 -17105.704,E2 -17105.704} C_VEL
LIN {X 0,Y 283.281,Z 573.055,A -85,B 0,C 180,E1 -17108.202,E2 -17108.202} C_VEL
LIN {X 0,Y 283.95,Z 565.036,A -85,B 0,C 180,E1 -17110.698,E2 -17110.698} C_VEL
LIN {X 0,Y 284.751,Z 556.478,A -85,B 0,C 180,E1 -17112.835,E2 -17112.835} C_VEL
LIN {X 0,Y 285.915,Z 545.867,A -85,B 0,C 180,E1 -17114.958,E2 -17114.958} C_VEL
LIN {X 0,Y 287.023,Z 536.197,A -85,B 0,C 180,E1 -17116.538,E2 -17116.538} C_VEL
LIN {X 0,Y 287.903,Z 525.253,A -85,B 0,C 180,E1 -17118.013,E2 -17118.013} C_VEL
LIN {X 0,Y 288.684,Z 516.455,A -85,B 0,C 180,E1 -17119.003,E2 -17119.003} C_VEL
LIN {X 0,Y 288.131,Z 511.699,A -85,B 0,C 180,E1 -17119.504,E2 -17119.504} C_VEL
LIN {X 0,Y 285.557,Z 498.302,A -85,B 0,C 180,E1 -17120.732,E2 -17120.732} C_VEL
LIN {X 0,Y 282.979,Z 484.536,A -85,B 0,C 180,E1 -17121.704,E2 -17121.704} C_VEL
LIN {X 0,Y 282.921,Z 484.131,A -85,B 0,C 180,E1 -17121.756,E2 -17121.756} C_VEL
LIN {X 0,Y 283.029,Z 481.339,A -85,B 0,C 180,E1 -17124.97,E2 -17124.97} C_VEL
LIN {X 0,Y 283.396,Z 481.186,A -85,B 0,C 180,E1 -17128.112,E2 -17128.112} C_VEL
LIN {X 0,Y 283.733,Z 481.139,A -85,B 0,C 180,E1 -17131.344,E2 -17131.344} C_VEL
LIN {X 0,Y 284.129,Z 481.09,A -85,B 0,C 180,E1 -17135.287,E2 -17135.287} C_VEL
LIN {X 0,Y 284.27,Z 481.077,A -85,B 0,C 180,E1 -17138.176,E2 -17138.176} C_VEL
LIN {X 0,Y 284.276,Z 481.072,A -85,B 0,C 180,E1 -17141.876,E2 -17141.876} C_VEL
LIN {X 0,Y 284.26,Z 481.078,A -85,B 0,C 180,E1 -17146.19,E2 -17146.19} C_VEL
LIN {X 0,Y 284.311,Z 481.07,A -85,B 0,C 180,E1 -17150.024,E2 -17150.024} C_VEL
LIN {X 0,Y 284.341,Z 481.064,A -85,B 0,C 180,E1 -17153.615,E2 -17153.615} C_VEL
LIN {X 0,Y 284.312,Z 481.067,A -85,B 0,C 180,E1 -17157.19,E2 -17157.19} C_VEL
LIN {X 0,Y 284.36,Z 481.064,A -85,B 0,C 180,E1 -17160.376,E2 -17160.376} C_VEL
LIN {X 0,Y 284.381,Z 481.06,A -85,B 0,C 180,E1 -17163.586,E2 -17163.586} C_VEL
LIN {X 0,Y 284.371,Z 481.06,A -85,B 0,C 180,E1 -17166.707,E2 -17166.707} C_VEL
LIN {X 0,Y 284.408,Z 481.055,A -85,B 0,C 180,E1 -17171.262,E2 -17171.262} C_VEL
LIN {X 0,Y 284.497,Z 481.046,A -85,B 0,C 180,E1 -17174.459,E2 -17174.459} C_VEL
LIN {X 0,Y 284.492,Z 481.045,A -85,B 0,C 180,E1 -17178.601,E2 -17178.601} C_VEL
LIN {X 0,Y 284.643,Z 481.027,A -85,B 0,C 180,E1 -17181.48,E2 -17181.48} C_VEL
LIN {X 0,Y 284.601,Z 481.033,A -85,B 0,C 180,E1 -17184.331,E2 -17184.331} C_VEL
LIN {X 0,Y 284.859,Z 481,A -85,B 0,C 180,E1 -17188.586,E2 -17188.586} C_VEL
LIN {X 0,Y 284.86,Z 481,A -85,B 0,C 180,E1 -17191.413,E2 -17191.413} C_VEL
LIN {X 0,Y 284.659,Z 481.024,A -85,B 0,C 180,E1 -17197.091,E2 -17197.091} C_VEL
LIN {X 0,Y 284.522,Z 481.046,A -85,B 0,C 180,E1 -17199.957,E2 -17199.957} C_VEL
LIN {X 0,Y 284.486,Z 481.047,A -85,B 0,C 180,E1 -17204.302,E2 -17204.302} C_VEL
LIN {X 0,Y 284.43,Z 481.053,A -85,B 0,C 180,E1 -17207.248,E2 -17207.248} C_VEL
LIN {X 0,Y 284.382,Z 481.06,A -85,B 0,C 180,E1 -17210.242,E2 -17210.242} C_VEL
LIN {X 0,Y 284.373,Z 481.064,A -85,B 0,C 180,E1 -17213.875,E2 -17213.875} C_VEL
LIN {X 0,Y 284.398,Z 481.057,A -85,B 0,C 180,E1 -17217.172,E2 -17217.172} C_VEL
LIN {X 0,Y 284.297,Z 481.069,A -85,B 0,C 180,E1 -17221.274,E2 -17221.274} C_VEL
LIN {X 0,Y 284.364,Z 481.062,A -85,B 0,C 180,E1 -17225.353,E2 -17225.353} C_VEL
LIN {X 0,Y 284.326,Z 481.066,A -85,B 0,C 180,E1 -17228.167,E2 -17228.167} C_VEL
LIN {X 0,Y 284.271,Z 481.074,A -85,B 0,C 180,E1 -17232.124,E2 -17232.124} C_VEL
LIN {X 0,Y 284.257,Z 481.075,A -85,B 0,C 180,E1 -17236.189,E2 -17236.189} C_VEL
LIN {X 0,Y 284.308,Z 481.07,A -85,B 0,C 180,E1 -17240.023,E2 -17240.023} C_VEL
LIN {X 0,Y 284.336,Z 481.069,A -85,B 0,C 180,E1 -17243.614,E2 -17243.614} C_VEL
LIN {X 0,Y 284.309,Z 481.068,A -85,B 0,C 180,E1 -17247.189,E2 -17247.189} C_VEL
LIN {X 0,Y 284.36,Z 481.061,A -85,B 0,C 180,E1 -17250.376,E2 -17250.376} C_VEL
LIN {X 0,Y 284.379,Z 481.063,A -85,B 0,C 180,E1 -17253.586,E2 -17253.586} C_VEL
LIN {X 0,Y 284.367,Z 481.059,A -85,B 0,C 180,E1 -17256.707,E2 -17256.707} C_VEL
LIN {X 0,Y 284.405,Z 481.058,A -85,B 0,C 180,E1 -17261.261,E2 -17261.261} C_VEL
LIN {X 0,Y 284.493,Z 481.043,A -85,B 0,C 180,E1 -17264.459,E2 -17264.459} C_VEL
LIN {X 0,Y 284.489,Z 481.045,A -85,B 0,C 180,E1 -17268.601,E2 -17268.601} C_VEL
LIN {X 0,Y 284.66,Z 481.028,A -85,B 0,C 180,E1 -17271.481,E2 -17271.481} C_VEL
LIN {X 0,Y 284.602,Z 481.03,A -85,B 0,C 180,E1 -17274.331,E2 -17274.331} C_VEL
LIN {X 0,Y 284.857,Z 480.999,A -85,B 0,C 180,E1 -17278.586,E2 -17278.586} C_VEL
LIN {X 0,Y 284.856,Z 481.003,A -85,B 0,C 180,E1 -17281.413,E2 -17281.413} C_VEL
LIN {X 0,Y 284.699,Z 481.021,A -85,B 0,C 180,E1 -17287.09,E2 -17287.09} C_VEL
LIN {X 0,Y 284.567,Z 481.035,A -85,B 0,C 180,E1 -17289.955,E2 -17289.955} C_VEL
LIN {X 0,Y 284.482,Z 481.046,A -85,B 0,C 180,E1 -17294.303,E2 -17294.303} C_VEL
LIN {X 0,Y 284.464,Z 481.049,A -85,B 0,C 180,E1 -17296.008,E2 -17296.008} C_VEL
LIN {X 0,Y 283.714,Z 481.145,A -85,B 0,C 180,E1 -17297.19,E2 -17297.19} C_VEL
LIN {X 0,Y 280.77,Z 481.51,A -85,B 0,C 180,E1 -17299.112,E2 -17299.112} C_VEL
LIN {X 0,Y 278.342,Z 481.81,A -85,B 0,C 180,E1 -17300.675,E2 -17300.675} C_VEL
LIN {X 0,Y 277.343,Z 481.936,A -85,B 0,C 180,E1 -17301.887,E2 -17301.887} C_VEL
LIN {X 0,Y 277.283,Z 481.942,A -85,B 0,C 180,E1 -17302.297,E2 -17302.297} C_VEL
LIN {X 0,Y 277.311,Z 481.942,A -85,B 0,C 180,E1 -17305.521,E2 -17305.521} C_VEL
LIN {X 0,Y 277.267,Z 481.944,A -85,B 0,C 180,E1 -17308.79,E2 -17308.79} C_VEL
LIN {X 0,Y 277.243,Z 481.948,A -85,B 0,C 180,E1 -17312.164,E2 -17312.164} C_VEL
LIN {X 0,Y 277.325,Z 481.938,A -85,B 0,C 180,E1 -17315.812,E2 -17315.812} C_VEL
LIN {X 0,Y 277.266,Z 481.949,A -85,B 0,C 180,E1 -17319.323,E2 -17319.323} C_VEL
LIN {X 0,Y 277.368,Z 482.024,A -85,B 0,C 180,E1 -17323.542,E2 -17323.542} C_VEL
LIN {X 0,Y 278.391,Z 487.779,A -85,B 0,C 180,E1 -17328.078,E2 -17328.078} C_VEL
LIN {X 0,Y 279.323,Z 493.121,A -85,B 0,C 180,E1 -17332.094,E2 -17332.094} C_VEL
LIN {X 0,Y 279.242,Z 496.68,A -85,B 0,C 180,E1 -17334.629,E2 -17334.629} C_VEL
LIN {X 0,Y 278.36,Z 501.524,A -85,B 0,C 180,E1 -17337.981,E2 -17337.981} C_VEL
LIN {X 0,Y 277.609,Z 506.306,A -85,B 0,C 180,E1 -17341.249,E2 -17341.249} C_VEL
LIN {X 0,Y 276.623,Z 513.366,A -85,B 0,C 180,E1 -17346.015,E2 -17346.015} C_VEL
LIN {X 0,Y 276.311,Z 516.036,A -85,B 0,C 180,E1 -17347.818,E2 -17347.818} C_VEL
LIN {X 0,Y 277.505,Z 531.093,A -85,B 0,C 180,E1 -17348.845,E2 -17348.845} C_VEL
LIN {X 0,Y 278.853,Z 545.073,A -85,B 0,C 180,E1 -17350.109,E2 -17350.109} C_VEL
LIN {X 0,Y 280.069,Z 557.477,A -85,B 0,C 180,E1 -17351.53,E2 -17351.53} C_VEL
LIN {X 0,Y 279.855,Z 563.109,A -85,B 0,C 180,E1 -17352.273,E2 -17352.273} C_VEL
LIN {X 0,Y 278.668,Z 573.747,A -85,B 0,C 180,E1 -17353.894,E2 -17353.894} C_VEL
LIN {X 0,Y 277.671,Z 583.452,A -85,B 0,C 180,E1 -17355.713,E2 -17355.713} C_VEL
LIN {X 0,Y 276.768,Z 592.909,A -85,B 0,C 180,E1 -17357.908,E2 -17357.908} C_VEL
LIN {X 0,Y 276.162,Z 600.567,A -85,B 0,C 180,E1 -17360.109,E2 -17360.109} C_VEL
LIN {X 0,Y 275.805,Z 607.581,A -85,B 0,C 180,E1 -17362.68,E2 -17362.68} C_VEL
LIN {X 0,Y 275.724,Z 612.228,A -85,B 0,C 180,E1 -17364.882,E2 -17364.882} C_VEL
LIN {X 0,Y 275.632,Z 615.698,A -85,B 0,C 180,E1 -17367.077,E2 -17367.077} C_VEL
LIN {X 0,Y 275.823,Z 617.466,A -85,B 0,C 180,E1 -17368.54,E2 -17368.54} C_VEL
LIN {X 0,Y 275.832,Z 618.719,A -85,B 0,C 180,E1 -17370,E2 -17370} C_VEL
LIN {X 0,Y 275.635,Z 619.518,A -85,B 0,C 180,E1 -17371.461,E2 -17371.461} C_VEL
LIN {X 0,Y 275.385,Z 619.928,A -85,B 0,C 180,E1 -17374.391,E2 -17374.391} C_VEL
LIN {X 0,Y 275.375,Z 619.518,A -85,B 0,C 180,E1 -17375.86,E2 -17375.86} C_VEL
LIN {X 0,Y 275.738,Z 617.51,A -85,B 0,C 180,E1 -17378.797,E2 -17378.797} C_VEL
LIN {X 0,Y 276.725,Z 613.993,A -85,B 0,C 180,E1 -17381.723,E2 -17381.723} C_VEL
LIN {X 0,Y 277.892,Z 610.251,A -85,B 0,C 180,E1 -17383.902,E2 -17383.902} C_VEL
LIN {X 0,Y 279.649,Z 605.582,A -85,B 0,C 180,E1 -17386.049,E2 -17386.049} C_VEL
LIN {X 0,Y 281.979,Z 598.919,A -85,B 0,C 180,E1 -17388.503,E2 -17388.503} C_VEL
LIN {X 0,Y 285.244,Z 590.484,A -85,B 0,C 180,E1 -17390.932,E2 -17390.932} C_VEL
LIN {X 0,Y 288.539,Z 581.862,A -85,B 0,C 180,E1 -17392.937,E2 -17392.937} C_VEL
LIN {X 0,Y 291.564,Z 573.452,A -85,B 0,C 180,E1 -17394.57,E2 -17394.57} C_VEL
LIN {X 0,Y 293.455,Z 564.763,A -85,B 0,C 180,E1 -17396.205,E2 -17396.205} C_VEL
LIN {X 0,Y 294.106,Z 556.24,A -85,B 0,C 180,E1 -17397.852,E2 -17397.852} C_VEL
LIN {X 0,Y 293.846,Z 546.613,A -85,B 0,C 180,E1 -17399.803,E2 -17399.803} C_VEL
LIN {X 0,Y 292.763,Z 537.314,A -85,B 0,C 180,E1 -17401.879,E2 -17401.879} C_VEL
LIN {X 0,Y 291.146,Z 528.368,A -85,B 0,C 180,E1 -17404.153,E2 -17404.153} C_VEL
LIN {X 0,Y 289.65,Z 522.165,A -85,B 0,C 180,E1 -17406.048,E2 -17406.048} C_VEL
LIN {X 0,Y 288.233,Z 516.627,A -85,B 0,C 180,E1 -17408.07,E2 -17408.07} C_VEL
LIN {X 0,Y 285.928,Z 511.032,A -85,B 0,C 180,E1 -17411.579,E2 -17411.579} C_VEL
LIN {X 0,Y 285.495,Z 508.471,A -85,B 0,C 180,E1 -17413.573,E2 -17413.573} C_VEL
LIN {X 0,Y 285.312,Z 507.374,A -85,B 0,C 180,E1 -17415.59,E2 -17415.59} C_VEL
LIN {X 0,Y 285.443,Z 507.627,A -85,B 0,C 180,E1 -17417.616,E2 -17417.616} C_VEL
LIN {X 0,Y 287.387,Z 509.553,A -85,B 0,C 180,E1 -17421.496,E2 -17421.496} C_VEL
LIN {X 0,Y 288.35,Z 510.17,A -85,B 0,C 180,E1 -17422.459,E2 -17422.459} C_VEL
LIN {X 0,Y 288.914,Z 511.736,A -85,B 0,C 180,E1 -17423.394,E2 -17423.394} C_VEL
LIN {X 0,Y 290.84,Z 514.423,A -85,B 0,C 180,E1 -17425.245,E2 -17425.245} C_VEL
LIN {X 0,Y 293.416,Z 519.689,A -85,B 0,C 180,E1 -17427.672,E2 -17427.672} C_VEL
LIN {X 0,Y 295.57,Z 524.834,A -85,B 0,C 180,E1 -17429.613,E2 -17429.613} C_VEL
LIN {X 0,Y 297.985,Z 533.343,A -85,B 0,C 180,E1 -17432.205,E2 -17432.205} C_VEL
LIN {X 0,Y 298.982,Z 539.527,A -85,B 0,C 180,E1 -17433.871,E2 -17433.871} C_VEL
LIN {X 0,Y 298.87,Z 541.297,A -85,B 0,C 180,E1 -17434.256,E2 -17434.256} C_VEL
LIN {X 0,Y 295.637,Z 550.351,A -85,B 0,C 180,E1 -17435.791,E2 -17435.791} C_VEL
LIN {X 0,Y 291.958,Z 559.629,A -85,B 0,C 180,E1 -17437.72,E2 -17437.72} C_VEL
LIN {X 0,Y 288.122,Z 568.544,A -85,B 0,C 180,E1 -17440.032,E2 -17440.032} C_VEL
LIN {X 0,Y 285.376,Z 574.669,A -85,B 0,C 180,E1 -17442.071,E2 -17442.071} C_VEL
LIN {X 0,Y 282.969,Z 579.721,A -85,B 0,C 180,E1 -17444.145,E2 -17444.145} C_VEL
LIN {X 0,Y 281,Z 583.704,A -85,B 0,C 180,E1 -17446.255,E2 -17446.255} C_VEL
LIN {X 0,Y 279.315,Z 586.735,A -85,B 0,C 180,E1 -17448.388,E2 -17448.388} C_VEL
LIN {X 0,Y 278.335,Z 588.419,A -85,B 0,C 180,E1 -17449.985,E2 -17449.985} C_VEL
LIN {X 0,Y 276.866,Z 590.166,A -85,B 0,C 180,E1 -17452.709,E2 -17452.709} C_VEL
LIN {X 0,Y 276.231,Z 590.517,A -85,B 0,C 180,E1 -17455.623,E2 -17455.623} C_VEL
LIN {X 0,Y 275.899,Z 590.099,A -85,B 0,C 180,E1 -17457.08,E2 -17457.08} C_VEL
LIN {X 0,Y 275.536,Z 588.089,A -85,B 0,C 180,E1 -17460,E2 -17460} C_VEL
LIN {X 0,Y 275.517,Z 585.51,A -85,B 0,C 180,E1 -17462.193,E2 -17462.193} C_VEL
LIN {X 0,Y 275.677,Z 581.96,A -85,B 0,C 180,E1 -17464.387,E2 -17464.387} C_VEL
LIN {X 0,Y 275.944,Z 576.565,A -85,B 0,C 180,E1 -17466.904,E2 -17466.904} C_VEL
LIN {X 0,Y 276.364,Z 570.382,A -85,B 0,C 180,E1 -17469.146,E2 -17469.146} C_VEL
LIN {X 0,Y 277.056,Z 562.903,A -85,B 0,C 180,E1 -17471.338,E2 -17471.338} C_VEL
LIN {X 0,Y 277.98,Z 553.765,A -85,B 0,C 180,E1 -17473.525,E2 -17473.525} C_VEL
LIN {X 0,Y 279.059,Z 543.444,A -85,B 0,C 180,E1 -17475.521,E2 -17475.521} C_VEL
LIN {X 0,Y 280.207,Z 533.256,A -85,B 0,C 180,E1 -17477.14,E2 -17477.14} C_VEL
LIN {X 0,Y 281.174,Z 522.404,A -85,B 0,C 180,E1 -17478.568,E2 -17478.568} C_VEL
LIN {X 0,Y 281.649,Z 515.736,A -85,B 0,C 180,E1 -17479.307,E2 -17479.307} C_VEL
LIN {X 0,Y 279.173,Z 502.511,A -85,B 0,C 180,E1 -17480.637,E2 -17480.637} C_VEL
LIN {X 0,Y 276.47,Z 488.131,A -85,B 0,C 180,E1 -17481.749,E2 -17481.749} C_VEL
LIN {X 0,Y 275.853,Z 484.565,A -85,B 0,C 180,E1 -17481.975,E2 -17481.975} C_VEL
LIN {X 0,Y 275.912,Z 482.768,A -85,B 0,C 180,E1 -17484.052,E2 -17484.052} C_VEL
LIN {X 0,Y 276.039,Z 482.102,A -85,B 0,C 180,E1 -17485.647,E2 -17485.647} C_VEL
LIN {X 0,Y 276.452,Z 482.047,A -85,B 0,C 180,E1 -17488.883,E2 -17488.883} C_VEL
LIN {X 0,Y 276.882,Z 481.991,A -85,B 0,C 180,E1 -17493.109,E2 -17493.109} C_VEL
LIN {X 0,Y 277.113,Z 481.965,A -85,B 0,C 180,E1 -17495.75,E2 -17495.75} C_VEL
LIN {X 0,Y 277.224,Z 481.95,A -85,B 0,C 180,E1 -17499.331,E2 -17499.331} C_VEL
LIN {X 0,Y 277.213,Z 481.951,A -85,B 0,C 180,E1 -17503.198,E2 -17503.198} C_VEL
LIN {X 0,Y 277.219,Z 481.951,A -85,B 0,C 180,E1 -17507.325,E2 -17507.325} C_VEL
LIN {X 0,Y 277.276,Z 481.944,A -85,B 0,C 180,E1 -17511.791,E2 -17511.791} C_VEL
LIN {X 0,Y 277.291,Z 481.946,A -85,B 0,C 180,E1 -17514.342,E2 -17514.342} C_VEL
LIN {X 0,Y 277.248,Z 481.949,A -85,B 0,C 180,E1 -17517.836,E2 -17517.836} C_VEL
LIN {X 0,Y 277.273,Z 481.943,A -85,B 0,C 180,E1 -17521.21,E2 -17521.21} C_VEL
LIN {X 0,Y 277.317,Z 481.941,A -85,B 0,C 180,E1 -17524.479,E2 -17524.479} C_VEL
LIN {X 0,Y 277.29,Z 481.942,A -85,B 0,C 180,E1 -17527.655,E2 -17527.655} C_VEL
LIN {X 0,Y 277.35,Z 481.935,A -85,B 0,C 180,E1 -17530.766,E2 -17530.766} C_VEL
LIN {X 0,Y 277.44,Z 481.923,A -85,B 0,C 180,E1 -17535.326,E2 -17535.326} C_VEL
LIN {X 0,Y 277.466,Z 481.922,A -85,B 0,C 180,E1 -17539.787,E2 -17539.787} C_VEL
LIN {X 0,Y 277.645,Z 481.898,A -85,B 0,C 180,E1 -17542.729,E2 -17542.729} C_VEL
LIN {X 0,Y 277.825,Z 481.876,A -85,B 0,C 180,E1 -17548.55,E2 -17548.55} C_VEL
LIN {X 0,Y 277.826,Z 481.876,A -85,B 0,C 180,E1 -17551.449,E2 -17551.449} C_VEL
LIN {X 0,Y 277.617,Z 481.901,A -85,B 0,C 180,E1 -17557.272,E2 -17557.272} C_VEL
LIN {X 0,Y 277.464,Z 481.922,A -85,B 0,C 180,E1 -17560.213,E2 -17560.213} C_VEL
LIN {X 0,Y 277.439,Z 481.923,A -85,B 0,C 180,E1 -17564.674,E2 -17564.674} C_VEL
LIN {X 0,Y 277.349,Z 481.935,A -85,B 0,C 180,E1 -17569.233,E2 -17569.233} C_VEL
LIN {X 0,Y 277.323,Z 481.94,A -85,B 0,C 180,E1 -17574.17,E2 -17574.17} C_VEL
LIN {X 0,Y 277.327,Z 481.94,A -85,B 0,C 180,E1 -17577.504,E2 -17577.504} C_VEL
LIN {X 0,Y 277.275,Z 481.943,A -85,B 0,C 180,E1 -17580.481,E2 -17580.481} C_VEL
LIN {X 0,Y 277.257,Z 481.95,A -85,B 0,C 180,E1 -17583.894,E2 -17583.894} C_VEL
LIN {X 0,Y 277.284,Z 481.945,A -85,B 0,C 180,E1 -17587.466,E2 -17587.466} C_VEL
LIN {X 0,Y 277.212,Z 481.952,A -85,B 0,C 180,E1 -17591.236,E2 -17591.236} C_VEL
LIN {X 0,Y 277.203,Z 481.954,A -85,B 0,C 180,E1 -17595.226,E2 -17595.226} C_VEL
LIN {X 0,Y 277.224,Z 481.952,A -85,B 0,C 180,E1 -17599.511,E2 -17599.511} C_VEL
LIN {X 0,Y 277.273,Z 481.944,A -85,B 0,C 180,E1 -17602.531,E2 -17602.531} C_VEL
LIN {X 0,Y 277.249,Z 481.947,A -85,B 0,C 180,E1 -17606.104,E2 -17606.104} C_VEL
LIN {X 0,Y 277.262,Z 481.948,A -85,B 0,C 180,E1 -17609.538,E2 -17609.538} C_VEL
LIN {X 0,Y 277.36,Z 481.933,A -85,B 0,C 180,E1 -17612.864,E2 -17612.864} C_VEL
LIN {X 0,Y 277.33,Z 481.937,A -85,B 0,C 180,E1 -17616.079,E2 -17616.079} C_VEL
LIN {X 0,Y 277.346,Z 481.935,A -85,B 0,C 180,E1 -17620.766,E2 -17620.766} C_VEL
LIN {X 0,Y 277.435,Z 481.925,A -85,B 0,C 180,E1 -17625.325,E2 -17625.325} C_VEL
LIN {X 0,Y 277.507,Z 481.918,A -85,B 0,C 180,E1 -17629.788,E2 -17629.788} C_VEL
LIN {X 0,Y 277.654,Z 481.896,A -85,B 0,C 180,E1 -17632.729,E2 -17632.729} C_VEL
LIN {X 0,Y 277.822,Z 481.875,A -85,B 0,C 180,E1 -17638.55,E2 -17638.55} C_VEL
LIN {X 0,Y 277.822,Z 481.879,A -85,B 0,C 180,E1 -17641.449,E2 -17641.449} C_VEL
LIN {X 0,Y 277.654,Z 481.9,A -85,B 0,C 180,E1 -17647.271,E2 -17647.271} C_VEL
LIN {X 0,Y 277.507,Z 481.914,A -85,B 0,C 180,E1 -17650.211,E2 -17650.211} C_VEL
LIN {X 0,Y 277.435,Z 481.924,A -85,B 0,C 180,E1 -17654.674,E2 -17654.674} C_VEL
LIN {X 0,Y 277.345,Z 481.938,A -85,B 0,C 180,E1 -17659.234,E2 -17659.234} C_VEL
LIN {X 0,Y 277.283,Z 481.942,A -85,B 0,C 180,E1 -17662.297,E2 -17662.297} C_VEL
LIN {X 0,Y 276.671,Z 482.024,A -85,B 0,C 180,E1 -17663.51,E2 -17663.51} C_VEL
LIN {X 0,Y 273.837,Z 482.377,A -85,B 0,C 180,E1 -17665.485,E2 -17665.485} C_VEL
LIN {X 0,Y 271.381,Z 482.68,A -85,B 0,C 180,E1 -17667.09,E2 -17667.09} C_VEL
LIN {X 0,Y 270.301,Z 482.811,A -85,B 0,C 180,E1 -17668.335,E2 -17668.335} C_VEL
LIN {X 0,Y 270.202,Z 482.822,A -85,B 0,C 180,E1 -17668.757,E2 -17668.757} C_VEL
LIN {X 0,Y 270.203,Z 482.828,A -85,B 0,C 180,E1 -17673.107,E2 -17673.107} C_VEL
LIN {X 0,Y 270.24,Z 482.82,A -85,B 0,C 180,E1 -17676.737,E2 -17676.737} C_VEL
LIN {X 0,Y 270.266,Z 482.82,A -85,B 0,C 180,E1 -17681.052,E2 -17681.052} C_VEL
LIN {X 0,Y 270.348,Z 482.971,A -85,B 0,C 180,E1 -17683.507,E2 -17683.507} C_VEL
LIN {X 0,Y 271.224,Z 488.071,A -85,B 0,C 180,E1 -17687.646,E2 -17687.646} C_VEL
LIN {X 0,Y 272.192,Z 493.317,A -85,B 0,C 180,E1 -17691.707,E2 -17691.707} C_VEL
LIN {X 0,Y 272.303,Z 495.843,A -85,B 0,C 180,E1 -17693.586,E2 -17693.586} C_VEL
LIN {X 0,Y 271.882,Z 498.933,A -85,B 0,C 180,E1 -17695.81,E2 -17695.81} C_VEL
LIN {X 0,Y 270.69,Z 505.488,A -85,B 0,C 180,E1 -17700.442,E2 -17700.442} C_VEL
LIN {X 0,Y 269.778,Z 511.357,A -85,B 0,C 180,E1 -17704.543,E2 -17704.543} C_VEL
LIN {X 0,Y 269.255,Z 515.766,A -85,B 0,C 180,E1 -17707.61,E2 -17707.61} C_VEL
LIN {X 0,Y 270.317,Z 529.827,A -85,B 0,C 180,E1 -17708.555,E2 -17708.555} C_VEL
LIN {X 0,Y 271.613,Z 544.025,A -85,B 0,C 180,E1 -17709.855,E2 -17709.855} C_VEL
LIN {X 0,Y 272.811,Z 555.82,A -85,B 0,C 180,E1 -17711.215,E2 -17711.215} C_VEL
LIN {X 0,Y 273.055,Z 560.36,A -85,B 0,C 180,E1 -17711.816,E2 -17711.816} C_VEL
LIN {X 0,Y 271.836,Z 571.297,A -85,B 0,C 180,E1 -17713.478,E2 -17713.478} C_VEL
LIN {X 0,Y 270.793,Z 581.328,A -85,B 0,C 180,E1 -17715.342,E2 -17715.342} C_VEL
LIN {X 0,Y 269.947,Z 589.634,A -85,B 0,C 180,E1 -17717.215,E2 -17717.215} C_VEL
LIN {X 0,Y 269.217,Z 597.789,A -85,B 0,C 180,E1 -17719.471,E2 -17719.471} C_VEL
LIN {X 0,Y 268.832,Z 604.389,A -85,B 0,C 180,E1 -17721.733,E2 -17721.733} C_VEL
LIN {X 0,Y 268.667,Z 609.639,A -85,B 0,C 180,E1 -17723.994,E2 -17723.994} C_VEL
LIN {X 0,Y 268.605,Z 613.658,A -85,B 0,C 180,E1 -17726.25,E2 -17726.25} C_VEL
LIN {X 0,Y 268.768,Z 616.571,A -85,B 0,C 180,E1 -17728.502,E2 -17728.502} C_VEL
LIN {X 0,Y 268.779,Z 617.949,A -85,B 0,C 180,E1 -17730,E2 -17730} C_VEL
LIN {X 0,Y 268.568,Z 618.848,A -85,B 0,C 180,E1 -17731.5,E2 -17731.5} C_VEL
LIN {X 0,Y 268.308,Z 619.422,A -85,B 0,C 180,E1 -17734.507,E2 -17734.507} C_VEL
LIN {X 0,Y 268.408,Z 618.444,A -85,B 0,C 180,E1 -17737.523,E2 -17737.523} C_VEL
LIN {X 0,Y 269.156,Z 615.883,A -85,B 0,C 180,E1 -17740.532,E2 -17740.532} C_VEL
LIN {X 0,Y 270.476,Z 611.811,A -85,B 0,C 180,E1 -17743.524,E2 -17743.524} C_VEL
LIN {X 0,Y 272.246,Z 607.669,A -85,B 0,C 180,E1 -17745.727,E2 -17745.727} C_VEL
LIN {X 0,Y 274.747,Z 601.202,A -85,B 0,C 180,E1 -17748.438,E2 -17748.438} C_VEL
LIN {X 0,Y 277.672,Z 594.147,A -85,B 0,C 180,E1 -17750.754,E2 -17750.754} C_VEL
LIN {X 0,Y 281.578,Z 584.952,A -85,B 0,C 180,E1 -17753.149,E2 -17753.149} C_VEL
LIN {X 0,Y 285.363,Z 575.518,A -85,B 0,C 180,E1 -17755.141,E2 -17755.141} C_VEL
LIN {X 0,Y 287.577,Z 566.826,A -85,B 0,C 180,E1 -17756.88,E2 -17756.88} C_VEL
LIN {X 0,Y 288.538,Z 557.888,A -85,B 0,C 180,E1 -17758.734,E2 -17758.734} C_VEL
LIN {X 0,Y 288.518,Z 548.679,A -85,B 0,C 180,E1 -17760.767,E2 -17760.767} C_VEL
LIN {X 0,Y 287.621,Z 538.883,A -85,B 0,C 180,E1 -17763.17,E2 -17763.17} C_VEL
LIN {X 0,Y 286.656,Z 532.307,A -85,B 0,C 180,E1 -17765.029,E2 -17765.029} C_VEL
LIN {X 0,Y 286.104,Z 528.726,A -85,B 0,C 180,E1 -17766.125,E2 -17766.125} C_VEL
LIN {X 0,Y 285.003,Z 523.572,A -85,B 0,C 180,E1 -17768.06,E2 -17768.06} C_VEL
LIN {X 0,Y 283.804,Z 520.36,A -85,B 0,C 180,E1 -17769.855,E2 -17769.855} C_VEL
LIN {X 0,Y 282.823,Z 515.835,A -85,B 0,C 180,E1 -17772.988,E2 -17772.988} C_VEL
LIN {X 0,Y 282.693,Z 514.739,A -85,B 0,C 180,E1 -17774.116,E2 -17774.116} C_VEL
LIN {X 0,Y 282.632,Z 513.889,A -85,B 0,C 180,E1 -17776.148,E2 -17776.148} C_VEL
LIN {X 0,Y 282.808,Z 514.414,A -85,B 0,C 180,E1 -17778.205,E2 -17778.205} C_VEL
LIN {X 0,Y 284.79,Z 516.249,A -85,B 0,C 180,E1 -17781.907,E2 -17781.907} C_VEL
LIN {X 0,Y 286.393,Z 519,A -85,B 0,C 180,E1 -17784.078,E2 -17784.078} C_VEL
LIN {X 0,Y 288.091,Z 522.404,A -85,B 0,C 180,E1 -17786.041,E2 -17786.041} C_VEL
LIN {X 0,Y 289.91,Z 526.862,A -85,B 0,C 180,E1 -17788.046,E2 -17788.046} C_VEL
LIN {X 0,Y 291.699,Z 532.6,A -85,B 0,C 180,E1 -17790.154,E2 -17790.154} C_VEL
LIN {X 0,Y 292.944,Z 538.667,A -85,B 0,C 180,E1 -17792.079,E2 -17792.079} C_VEL
LIN {X 0,Y 293.474,Z 543.092,A -85,B 0,C 180,E1 -17793.342,E2 -17793.342} C_VEL
LIN {X 0,Y 291.586,Z 548.406,A -85,B 0,C 180,E1 -17794.288,E2 -17794.288} C_VEL
LIN {X 0,Y 286.997,Z 559.502,A -85,B 0,C 180,E1 -17796.551,E2 -17796.551} C_VEL
LIN {X 0,Y 283.416,Z 567.25,A -85,B 0,C 180,E1 -17798.546,E2 -17798.546} C_VEL
LIN {X 0,Y 280.71,Z 572.741,A -85,B 0,C 180,E1 -17800.246,E2 -17800.246} C_VEL
LIN {X 0,Y 277.92,Z 578.21,A -85,B 0,C 180,E1 -17802.335,E2 -17802.335} C_VEL
LIN {X 0,Y 274.876,Z 583.82,A -85,B 0,C 180,E1 -17805.186,E2 -17805.186} C_VEL
LIN {X 0,Y 273.496,Z 586.06,A -85,B 0,C 180,E1 -17806.628,E2 -17806.628} C_VEL
LIN {X 0,Y 271.515,Z 589.193,A -85,B 0,C 180,E1 -17809.561,E2 -17809.561} C_VEL
LIN {X 0,Y 269.87,Z 590.868,A -85,B 0,C 180,E1 -17812.519,E2 -17812.519} C_VEL
LIN {X 0,Y 269.481,Z 591.107,A -85,B 0,C 180,E1 -17814.012,E2 -17814.012} C_VEL
LIN {X 0,Y 269.163,Z 590.951,A -85,B 0,C 180,E1 -17815.508,E2 -17815.508} C_VEL
LIN {X 0,Y 268.581,Z 589.527,A -85,B 0,C 180,E1 -17818.501,E2 -17818.501} C_VEL
LIN {X 0,Y 268.449,Z 588.226,A -85,B 0,C 180,E1 -17820,E2 -17820} C_VEL
LIN {X 0,Y 268.442,Z 585.476,A -85,B 0,C 180,E1 -17822.251,E2 -17822.251} C_VEL
LIN {X 0,Y 268.578,Z 581.74,A -85,B 0,C 180,E1 -17824.503,E2 -17824.503} C_VEL
LIN {X 0,Y 268.863,Z 576.411,A -85,B 0,C 180,E1 -17826.964,E2 -17826.964} C_VEL
LIN {X 0,Y 269.341,Z 569.746,A -85,B 0,C 180,E1 -17829.386,E2 -17829.386} C_VEL
LIN {X 0,Y 270.065,Z 562.056,A -85,B 0,C 180,E1 -17831.636,E2 -17831.636} C_VEL
LIN {X 0,Y 271.014,Z 552.567,A -85,B 0,C 180,E1 -17833.88,E2 -17833.88} C_VEL
LIN {X 0,Y 272.111,Z 541.922,A -85,B 0,C 180,E1 -17835.928,E2 -17835.928} C_VEL
LIN {X 0,Y 273.213,Z 532.624,A -85,B 0,C 180,E1 -17837.4,E2 -17837.4} C_VEL
LIN {X 0,Y 274.251,Z 521.359,A -85,B 0,C 180,E1 -17838.876,E2 -17838.876} C_VEL
LIN {X 0,Y 274.575,Z 516.434,A -85,B 0,C 180,E1 -17839.436,E2 -17839.436} C_VEL
LIN {X 0,Y 272.117,Z 503.255,A -85,B 0,C 180,E1 -17840.807,E2 -17840.807} C_VEL
LIN {X 0,Y 269.521,Z 489.266,A -85,B 0,C 180,E1 -17841.935,E2 -17841.935} C_VEL
LIN {X 0,Y 268.808,Z 484.925,A -85,B 0,C 180,E1 -17842.242,E2 -17842.242} C_VEL
LIN {X 0,Y 268.87,Z 482.995,A -85,B 0,C 180,E1 -17844.723,E2 -17844.723} C_VEL
LIN {X 0,Y 269.278,Z 482.945,A -85,B 0,C 180,E1 -17848.021,E2 -17848.021} C_VEL
LIN {X 0,Y 269.625,Z 482.896,A -85,B 0,C 180,E1 -17851.421,E2 -17851.421} C_VEL
LIN {X 0,Y 269.974,Z 482.853,A -85,B 0,C 180,E1 -17854.94,E2 -17854.94} C_VEL
LIN {X 0,Y 270.171,Z 482.83,A -85,B 0,C 180,E1 -17858.702,E2 -17858.702} C_VEL
LIN {X 0,Y 270.176,Z 482.83,A -85,B 0,C 180,E1 -17862.558,E2 -17862.558} C_VEL
LIN {X 0,Y 270.169,Z 482.83,A -85,B 0,C 180,E1 -17866.751,E2 -17866.751} C_VEL
LIN {X 0,Y 270.226,Z 482.82,A -85,B 0,C 180,E1 -17871.283,E2 -17871.283} C_VEL
LIN {X 0,Y 270.207,Z 482.824,A -85,B 0,C 180,E1 -17875.095,E2 -17875.095} C_VEL
LIN {X 0,Y 270.205,Z 482.823,A -85,B 0,C 180,E1 -17879.131,E2 -17879.131} C_VEL
LIN {X 0,Y 270.268,Z 482.821,A -85,B 0,C 180,E1 -17882.146,E2 -17882.146} C_VEL
LIN {X 0,Y 270.282,Z 482.815,A -85,B 0,C 180,E1 -17885.519,E2 -17885.519} C_VEL
LIN {X 0,Y 270.306,Z 482.815,A -85,B 0,C 180,E1 -17890.244,E2 -17890.244} C_VEL
LIN {X 0,Y 270.408,Z 482.799,A -85,B 0,C 180,E1 -17894.935,E2 -17894.935} C_VEL
LIN {X 0,Y 270.418,Z 482.799,A -85,B 0,C 180,E1 -17899.518,E2 -17899.518} C_VEL
LIN {X 0,Y 270.603,Z 482.776,A -85,B 0,C 180,E1 -17902.538,E2 -17902.538} C_VEL
LIN {X 0,Y 270.791,Z 482.753,A -85,B 0,C 180,E1 -17908.512,E2 -17908.512} C_VEL
LIN {X 0,Y 270.792,Z 482.753,A -85,B 0,C 180,E1 -17911.487,E2 -17911.487} C_VEL
LIN {X 0,Y 270.576,Z 482.779,A -85,B 0,C 180,E1 -17917.462,E2 -17917.462} C_VEL
LIN {X 0,Y 270.417,Z 482.799,A -85,B 0,C 180,E1 -17920.482,E2 -17920.482} C_VEL
LIN {X 0,Y 270.407,Z 482.799,A -85,B 0,C 180,E1 -17925.064,E2 -17925.064} C_VEL
LIN {X 0,Y 270.305,Z 482.816,A -85,B 0,C 180,E1 -17929.755,E2 -17929.755} C_VEL
LIN {X 0,Y 270.277,Z 482.816,A -85,B 0,C 180,E1 -17934.585,E2 -17934.585} C_VEL
LIN {X 0,Y 270.273,Z 482.82,A -85,B 0,C 180,E1 -17937.908,E2 -17937.908} C_VEL
LIN {X 0,Y 270.187,Z 482.826,A -85,B 0,C 180,E1 -17941.348,E2 -17941.348} C_VEL
LIN {X 0,Y 270.226,Z 482.822,A -85,B 0,C 180,E1 -17944.902,E2 -17944.902} C_VEL
LIN {X 0,Y 270.224,Z 482.821,A -85,B 0,C 180,E1 -17948.716,E2 -17948.716} C_VEL
LIN {X 0,Y 270.167,Z 482.83,A -85,B 0,C 180,E1 -17953.248,E2 -17953.248} C_VEL
LIN {X 0,Y 270.173,Z 482.83,A -85,B 0,C 180,E1 -17957.441,E2 -17957.441} C_VEL
LIN {X 0,Y 270.208,Z 482.826,A -85,B 0,C 180,E1 -17961.374,E2 -17961.374} C_VEL
LIN {X 0,Y 270.204,Z 482.825,A -85,B 0,C 180,E1 -17965.094,E2 -17965.094} C_VEL
LIN {X 0,Y 270.201,Z 482.825,A -85,B 0,C 180,E1 -17969.13,E2 -17969.13} C_VEL
LIN {X 0,Y 270.266,Z 482.818,A -85,B 0,C 180,E1 -17972.145,E2 -17972.145} C_VEL
LIN {X 0,Y 270.278,Z 482.818,A -85,B 0,C 180,E1 -17975.519,E2 -17975.519} C_VEL
LIN {X 0,Y 270.303,Z 482.813,A -85,B 0,C 180,E1 -17980.244,E2 -17980.244} C_VEL
LIN {X 0,Y 270.404,Z 482.798,A -85,B 0,C 180,E1 -17984.935,E2 -17984.935} C_VEL
LIN {X 0,Y 270.442,Z 482.8,A -85,B 0,C 180,E1 -17989.519,E2 -17989.519} C_VEL
LIN {X 0,Y 270.612,Z 482.772,A -85,B 0,C 180,E1 -17992.538,E2 -17992.538} C_VEL
LIN {X 0,Y 270.788,Z 482.752,A -85,B 0,C 180,E1 -17998.512,E2 -17998.512} C_VEL
LIN {X 0,Y 270.788,Z 482.755,A -85,B 0,C 180,E1 -18001.487,E2 -18001.487} C_VEL
LIN {X 0,Y 270.612,Z 482.779,A -85,B 0,C 180,E1 -18007.461,E2 -18007.461} C_VEL
LIN {X 0,Y 270.442,Z 482.793,A -85,B 0,C 180,E1 -18010.481,E2 -18010.481} C_VEL
LIN {X 0,Y 270.403,Z 482.802,A -85,B 0,C 180,E1 -18015.064,E2 -18015.064} C_VEL
LIN {X 0,Y 270.301,Z 482.813,A -85,B 0,C 180,E1 -18019.755,E2 -18019.755} C_VEL
LIN {X 0,Y 270.273,Z 482.816,A -85,B 0,C 180,E1 -18024.585,E2 -18024.585} C_VEL
LIN {X 0,Y 270.202,Z 482.822,A -85,B 0,C 180,E1 -18028.757,E2 -18028.757} C_VEL
LIN {X 0,Y 269.498,Z 482.914,A -85,B 0,C 180,E1 -18030,E2 -18030} C_VEL
LIN {X 0,Y 266.622,Z 483.271,A -85,B 0,C 180,E1 -18032.025,E2 -18032.025} C_VEL
LIN {X 0,Y 264.221,Z 483.572,A -85,B 0,C 180,E1 -18033.672,E2 -18033.672} C_VEL
LIN {X 0,Y 263.22,Z 483.696,A -85,B 0,C 180,E1 -18034.948,E2 -18034.948} C_VEL
LIN {X 0,Y 263.153,Z 483.699,A -85,B 0,C 180,E1 -18035.381,E2 -18035.381} C_VEL
LIN {X 0,Y 263.157,Z 483.706,A -85,B 0,C 180,E1 -18039.242,E2 -18039.242} C_VEL
LIN {X 0,Y 263.309,Z 483.798,A -85,B 0,C 180,E1 -18043.404,E2 -18043.404} C_VEL
LIN {X 0,Y 264.332,Z 489.758,A -85,B 0,C 180,E1 -18048.342,E2 -18048.342} C_VEL
LIN {X 0,Y 265.06,Z 493.676,A -85,B 0,C 180,E1 -18051.458,E2 -18051.458} C_VEL
LIN {X 0,Y 265.136,Z 497.454,A -85,B 0,C 180,E1 -18054.327,E2 -18054.327} C_VEL
LIN {X 0,Y 264.06,Z 503.001,A -85,B 0,C 180,E1 -18058.395,E2 -18058.395} C_VEL
LIN {X 0,Y 263.033,Z 509.327,A -85,B 0,C 180,E1 -18062.985,E2 -18062.985} C_VEL
LIN {X 0,Y 262.226,Z 515.382,A -85,B 0,C 180,E1 -18067.34,E2 -18067.34} C_VEL
LIN {X 0,Y 263.182,Z 529.349,A -85,B 0,C 180,E1 -18068.327,E2 -18068.327} C_VEL
LIN {X 0,Y 264.432,Z 543.517,A -85,B 0,C 180,E1 -18069.663,E2 -18069.663} C_VEL
LIN {X 0,Y 265.666,Z 555.528,A -85,B 0,C 180,E1 -18071.091,E2 -18071.091} C_VEL
LIN {X 0,Y 265.911,Z 560.814,A -85,B 0,C 180,E1 -18071.819,E2 -18071.819} C_VEL
LIN {X 0,Y 264.612,Z 572.066,A -85,B 0,C 180,E1 -18073.609,E2 -18073.609} C_VEL
LIN {X 0,Y 263.506,Z 582.757,A -85,B 0,C 180,E1 -18075.718,E2 -18075.718} C_VEL
LIN {X 0,Y 262.599,Z 592.173,A -85,B 0,C 180,E1 -18078.029,E2 -18078.029} C_VEL
LIN {X 0,Y 262.015,Z 599.78,A -85,B 0,C 180,E1 -18080.349,E2 -18080.349} C_VEL
LIN {X 0,Y 261.738,Z 604.931,A -85,B 0,C 180,E1 -18082.285,E2 -18082.285} C_VEL
LIN {X 0,Y 261.639,Z 610.335,A -85,B 0,C 180,E1 -18084.833,E2 -18084.833} C_VEL
LIN {X 0,Y 261.55,Z 613.719,A -85,B 0,C 180,E1 -18086.92,E2 -18086.92} C_VEL
LIN {X 0,Y 261.715,Z 615.648,A -85,B 0,C 180,E1 -18088.462,E2 -18088.462} C_VEL
LIN {X 0,Y 261.727,Z 617.113,A -85,B 0,C 180,E1 -18090,E2 -18090} C_VEL
LIN {X 0,Y 261.502,Z 618.134,A -85,B 0,C 180,E1 -18091.54,E2 -18091.54} C_VEL
LIN {X 0,Y 261.276,Z 618.729,A -85,B 0,C 180,E1 -18093.084,E2 -18093.084} C_VEL
LIN {X 0,Y 261.212,Z 618.859,A -85,B 0,C 180,E1 -18095.439,E2 -18095.439} C_VEL
LIN {X 0,Y 261.343,Z 618.116,A -85,B 0,C 180,E1 -18097.728,E2 -18097.728} C_VEL
LIN {X 0,Y 262.135,Z 615.836,A -85,B 0,C 180,E1 -18100.817,E2 -18100.817} C_VEL
LIN {X 0,Y 263.57,Z 611.996,A -85,B 0,C 180,E1 -18103.886,E2 -18103.886} C_VEL
LIN {X 0,Y 266.07,Z 606.602,A -85,B 0,C 180,E1 -18106.892,E2 -18106.892} C_VEL
LIN {X 0,Y 268.668,Z 600.594,A -85,B 0,C 180,E1 -18109.443,E2 -18109.443} C_VEL
LIN {X 0,Y 272.237,Z 592.916,A -85,B 0,C 180,E1 -18111.983,E2 -18111.983} C_VEL
LIN {X 0,Y 276.458,Z 583.701,A -85,B 0,C 180,E1 -18114.4,E2 -18114.4} C_VEL
LIN {X 0,Y 279.757,Z 575.966,A -85,B 0,C 180,E1 -18116.081,E2 -18116.081} C_VEL
LIN {X 0,Y 281.673,Z 569.328,A -85,B 0,C 180,E1 -18117.49,E2 -18117.49} C_VEL
LIN {X 0,Y 282.912,Z 561.214,A -85,B 0,C 180,E1 -18119.293,E2 -18119.293} C_VEL
LIN {X 0,Y 283.3,Z 552.297,A -85,B 0,C 180,E1 -18121.397,E2 -18121.397} C_VEL
LIN {X 0,Y 282.902,Z 543.164,A -85,B 0,C 180,E1 -18123.797,E2 -18123.797} C_VEL
LIN {X 0,Y 282.148,Z 535.369,A -85,B 0,C 180,E1 -18126.192,E2 -18126.192} C_VEL
LIN {X 0,Y 281.515,Z 531.501,A -85,B 0,C 180,E1 -18127.618,E2 -18127.618} C_VEL
LIN {X 0,Y 280.971,Z 527.941,A -85,B 0,C 180,E1 -18129.158,E2 -18129.158} C_VEL
LIN {X 0,Y 279.759,Z 522.777,A -85,B 0,C 180,E1 -18132.71,E2 -18132.71} C_VEL
LIN {X 0,Y 279.64,Z 520.897,A -85,B 0,C 180,E1 -18134.726,E2 -18134.726} C_VEL
LIN {X 0,Y 279.611,Z 520.522,A -85,B 0,C 180,E1 -18137.263,E2 -18137.263} C_VEL
LIN {X 0,Y 280.807,Z 522.016,A -85,B 0,C 180,E1 -18140.884,E2 -18140.884} C_VEL
LIN {X 0,Y 282.301,Z 524.276,A -85,B 0,C 180,E1 -18143.31,E2 -18143.31} C_VEL
LIN {X 0,Y 283.695,Z 527.194,A -85,B 0,C 180,E1 -18145.265,E2 -18145.265} C_VEL
LIN {X 0,Y 285.475,Z 532.174,A -85,B 0,C 180,E1 -18147.728,E2 -18147.728} C_VEL
LIN {X 0,Y 286.739,Z 536.852,A -85,B 0,C 180,E1 -18149.584,E2 -18149.584} C_VEL
LIN {X 0,Y 287.78,Z 543.795,A -85,B 0,C 180,E1 -18151.931,E2 -18151.931} C_VEL
LIN {X 0,Y 287.691,Z 547.026,A -85,B 0,C 180,E1 -18152.853,E2 -18152.853} C_VEL
LIN {X 0,Y 283.547,Z 556.547,A -85,B 0,C 180,E1 -18154.687,E2 -18154.687} C_VEL
LIN {X 0,Y 278.922,Z 566.047,A -85,B 0,C 180,E1 -18157.011,E2 -18157.011} C_VEL
LIN {X 0,Y 275.355,Z 572.796,A -85,B 0,C 180,E1 -18159.064,E2 -18159.064} C_VEL
LIN {X 0,Y 272.332,Z 578.265,A -85,B 0,C 180,E1 -18161.181,E2 -18161.181} C_VEL
LIN {X 0,Y 269.656,Z 582.77,A -85,B 0,C 180,E1 -18163.34,E2 -18163.34} C_VEL
LIN {X 0,Y 267.47,Z 586.255,A -85,B 0,C 180,E1 -18165.545,E2 -18165.545} C_VEL
LIN {X 0,Y 265.612,Z 588.858,A -85,B 0,C 180,E1 -18167.78,E2 -18167.78} C_VEL
LIN {X 0,Y 264.49,Z 590.272,A -85,B 0,C 180,E1 -18169.472,E2 -18169.472} C_VEL
LIN {X 0,Y 262.879,Z 591.519,A -85,B 0,C 180,E1 -18172.318,E2 -18172.318} C_VEL
LIN {X 0,Y 262.099,Z 591.368,A -85,B 0,C 180,E1 -18175.386,E2 -18175.386} C_VEL
LIN {X 0,Y 261.747,Z 590.745,A -85,B 0,C 180,E1 -18176.922,E2 -18176.922} C_VEL
LIN {X 0,Y 261.499,Z 589.71,A -85,B 0,C 180,E1 -18178.46,E2 -18178.46} C_VEL
LIN {X 0,Y 261.343,Z 586.438,A -85,B 0,C 180,E1 -18181.541,E2 -18181.541} C_VEL
LIN {X 0,Y 261.457,Z 582.864,A -85,B 0,C 180,E1 -18183.854,E2 -18183.854} C_VEL
LIN {X 0,Y 261.679,Z 577.658,A -85,B 0,C 180,E1 -18186.42,E2 -18186.42} C_VEL
LIN {X 0,Y 262.121,Z 571.3,A -85,B 0,C 180,E1 -18188.869,E2 -18188.869} C_VEL
LIN {X 0,Y 262.77,Z 563.857,A -85,B 0,C 180,E1 -18191.181,E2 -18191.181} C_VEL
LIN {X 0,Y 263.693,Z 554.787,A -85,B 0,C 180,E1 -18193.486,E2 -18193.486} C_VEL
LIN {X 0,Y 264.871,Z 544.595,A -85,B 0,C 180,E1 -18195.585,E2 -18195.585} C_VEL
LIN {X 0,Y 266.127,Z 533.569,A -85,B 0,C 180,E1 -18197.428,E2 -18197.428} C_VEL
LIN {X 0,Y 267.154,Z 522.012,A -85,B 0,C 180,E1 -18198.999,E2 -18198.999} C_VEL
LIN {X 0,Y 267.512,Z 517.134,A -85,B 0,C 180,E1 -18199.571,E2 -18199.571} C_VEL
LIN {X 0,Y 265.07,Z 504.061,A -85,B 0,C 180,E1 -18200.979,E2 -18200.979} C_VEL
LIN {X 0,Y 262.57,Z 490.318,A -85,B 0,C 180,E1 -18202.137,E2 -18202.137} C_VEL
LIN {X 0,Y 261.73,Z 485.311,A -85,B 0,C 180,E1 -18202.498,E2 -18202.498} C_VEL
LIN {X 0,Y 261.798,Z 483.879,A -85,B 0,C 180,E1 -18204.317,E2 -18204.317} C_VEL
LIN {X 0,Y 262.217,Z 483.825,A -85,B 0,C 180,E1 -18207.812,E2 -18207.812} C_VEL
LIN {X 0,Y 262.558,Z 483.776,A -85,B 0,C 180,E1 -18211.067,E2 -18211.067} C_VEL
LIN {X 0,Y 262.861,Z 483.741,A -85,B 0,C 180,E1 -18214.158,E2 -18214.158} C_VEL
LIN {X 0,Y 263.062,Z 483.716,A -85,B 0,C 180,E1 -18217.914,E2 -18217.914} C_VEL
LIN {X 0,Y 263.127,Z 483.706,A -85,B 0,C 180,E1 -18221.893,E2 -18221.893} C_VEL
LIN {X 0,Y 263.128,Z 483.71,A -85,B 0,C 180,E1 -18226.151,E2 -18226.151} C_VEL
LIN {X 0,Y 263.119,Z 483.71,A -85,B 0,C 180,E1 -18230.13,E2 -18230.13} C_VEL
LIN {X 0,Y 263.181,Z 483.702,A -85,B 0,C 180,E1 -18234.021,E2 -18234.021} C_VEL
LIN {X 0,Y 263.137,Z 483.706,A -85,B 0,C 180,E1 -18237.712,E2 -18237.712} C_VEL
LIN {X 0,Y 263.203,Z 483.698,A -85,B 0,C 180,E1 -18241.784,E2 -18241.784} C_VEL
LIN {X 0,Y 263.23,Z 483.693,A -85,B 0,C 180,E1 -18245.2,E2 -18245.2} C_VEL
LIN {X 0,Y 263.268,Z 483.689,A -85,B 0,C 180,E1 -18249.693,E2 -18249.693} C_VEL
LIN {X 0,Y 263.356,Z 483.678,A -85,B 0,C 180,E1 -18254.522,E2 -18254.522} C_VEL
LIN {X 0,Y 263.36,Z 483.677,A -85,B 0,C 180,E1 -18259.233,E2 -18259.233} C_VEL
LIN {X 0,Y 263.563,Z 483.654,A -85,B 0,C 180,E1 -18262.338,E2 -18262.338} C_VEL
LIN {X 0,Y 263.756,Z 483.629,A -85,B 0,C 180,E1 -18268.473,E2 -18268.473} C_VEL
LIN {X 0,Y 263.756,Z 483.629,A -85,B 0,C 180,E1 -18271.527,E2 -18271.527} C_VEL
LIN {X 0,Y 263.538,Z 483.657,A -85,B 0,C 180,E1 -18277.662,E2 -18277.662} C_VEL
LIN {X 0,Y 263.359,Z 483.677,A -85,B 0,C 180,E1 -18280.766,E2 -18280.766} C_VEL
LIN {X 0,Y 263.355,Z 483.679,A -85,B 0,C 180,E1 -18285.477,E2 -18285.477} C_VEL
LIN {X 0,Y 263.267,Z 483.689,A -85,B 0,C 180,E1 -18290.306,E2 -18290.306} C_VEL
LIN {X 0,Y 263.211,Z 483.696,A -85,B 0,C 180,E1 -18295.291,E2 -18295.291} C_VEL
LIN {X 0,Y 263.178,Z 483.699,A -85,B 0,C 180,E1 -18298.729,E2 -18298.729} C_VEL
LIN {X 0,Y 263.136,Z 483.706,A -85,B 0,C 180,E1 -18302.287,E2 -18302.287} C_VEL
LIN {X 0,Y 263.193,Z 483.701,A -85,B 0,C 180,E1 -18305.977,E2 -18305.977} C_VEL
LIN {X 0,Y 263.117,Z 483.71,A -85,B 0,C 180,E1 -18309.87,E2 -18309.87} C_VEL
LIN {X 0,Y 263.124,Z 483.709,A -85,B 0,C 180,E1 -18313.983,E2 -18313.983} C_VEL
LIN {X 0,Y 263.126,Z 483.705,A -85,B 0,C 180,E1 -18318.406,E2 -18318.406} C_VEL
LIN {X 0,Y 263.186,Z 483.7,A -85,B 0,C 180,E1 -18323.235,E2 -18323.235} C_VEL
LIN {X 0,Y 263.168,Z 483.702,A -85,B 0,C 180,E1 -18325.887,E2 -18325.887} C_VEL
LIN {X 0,Y 263.152,Z 483.706,A -85,B 0,C 180,E1 -18329.506,E2 -18329.506} C_VEL
LIN {X 0,Y 263.194,Z 483.698,A -85,B 0,C 180,E1 -18333.002,E2 -18333.002} C_VEL
LIN {X 0,Y 263.185,Z 483.698,A -85,B 0,C 180,E1 -18336.387,E2 -18336.387} C_VEL
LIN {X 0,Y 263.265,Z 483.693,A -85,B 0,C 180,E1 -18339.693,E2 -18339.693} C_VEL
LIN {X 0,Y 263.352,Z 483.676,A -85,B 0,C 180,E1 -18344.522,E2 -18344.522} C_VEL
LIN {X 0,Y 263.375,Z 483.678,A -85,B 0,C 180,E1 -18349.234,E2 -18349.234} C_VEL
LIN {X 0,Y 263.574,Z 483.649,A -85,B 0,C 180,E1 -18352.338,E2 -18352.338} C_VEL
LIN {X 0,Y 263.752,Z 483.628,A -85,B 0,C 180,E1 -18358.473,E2 -18358.473} C_VEL
LIN {X 0,Y 263.752,Z 483.631,A -85,B 0,C 180,E1 -18361.527,E2 -18361.527} C_VEL
LIN {X 0,Y 263.573,Z 483.653,A -85,B 0,C 180,E1 -18367.661,E2 -18367.661} C_VEL
LIN {X 0,Y 263.374,Z 483.674,A -85,B 0,C 180,E1 -18370.765,E2 -18370.765} C_VEL
LIN {X 0,Y 263.351,Z 483.683,A -85,B 0,C 180,E1 -18375.478,E2 -18375.478} C_VEL
LIN {X 0,Y 263.263,Z 483.688,A -85,B 0,C 180,E1 -18380.306,E2 -18380.306} C_VEL
LIN {X 0,Y 263.207,Z 483.701,A -85,B 0,C 180,E1 -18385.291,E2 -18385.291} C_VEL
LIN {X 0,Y 263.165,Z 483.7,A -85,B 0,C 180,E1 -18388.731,E2 -18388.731} C_VEL
LIN {X 0,Y 263.133,Z 483.706,A -85,B 0,C 180,E1 -18392.288,E2 -18392.288} C_VEL
LIN {X 0,Y 263.153,Z 483.699,A -85,B 0,C 180,E1 -18395.381,E2 -18395.381} C_VEL
LIN {X 0,Y 262.509,Z 483.784,A -85,B 0,C 180,E1 -18396.659,E2 -18396.659} C_VEL
LIN {X 0,Y 259.631,Z 484.142,A -85,B 0,C 180,E1 -18398.742,E2 -18398.742} C_VEL
LIN {X 0,Y 257.213,Z 484.443,A -85,B 0,C 180,E1 -18400.437,E2 -18400.437} C_VEL
LIN {X 0,Y 256.238,Z 484.566,A -85,B 0,C 180,E1 -18401.752,E2 -18401.752} C_VEL
LIN {X 0,Y 256.194,Z 484.57,A -85,B 0,C 180,E1 -18402.197,E2 -18402.197} C_VEL
LIN {X 0,Y 256.248,Z 484.609,A -85,B 0,C 180,E1 -18403.288,E2 -18403.288} C_VEL
LIN {X 0,Y 257.111,Z 489.596,A -85,B 0,C 180,E1 -18407.564,E2 -18407.564} C_VEL
LIN {X 0,Y 257.919,Z 494.008,A -85,B 0,C 180,E1 -18411.192,E2 -18411.192} C_VEL
LIN {X 0,Y 258.097,Z 497.704,A -85,B 0,C 180,E1 -18414.092,E2 -18414.092} C_VEL
LIN {X 0,Y 257.09,Z 502.773,A -85,B 0,C 180,E1 -18417.934,E2 -18417.934} C_VEL
LIN {X 0,Y 256.078,Z 508.451,A -85,B 0,C 180,E1 -18422.189,E2 -18422.189} C_VEL
LIN {X 0,Y 255.157,Z 515.197,A -85,B 0,C 180,E1 -18427.105,E2 -18427.105} C_VEL
LIN {X 0,Y 256.032,Z 528.169,A -85,B 0,C 180,E1 -18428.03,E2 -18428.03} C_VEL
LIN {X 0,Y 257.188,Z 541.49,A -85,B 0,C 180,E1 -18429.297,E2 -18429.297} C_VEL
LIN {X 0,Y 258.507,Z 555.228,A -85,B 0,C 180,E1 -18430.959,E2 -18430.959} C_VEL
LIN {X 0,Y 258.859,Z 560.417,A -85,B 0,C 180,E1 -18431.697,E2 -18431.697} C_VEL
LIN {X 0,Y 257.526,Z 571.729,A -85,B 0,C 180,E1 -18433.553,E2 -18433.553} C_VEL
LIN {X 0,Y 256.417,Z 582.326,A -85,B 0,C 180,E1 -18435.719,E2 -18435.719} C_VEL
LIN {X 0,Y 255.522,Z 591.673,A -85,B 0,C 180,E1 -18438.096,E2 -18438.096} C_VEL
LIN {X 0,Y 254.95,Z 599.251,A -85,B 0,C 180,E1 -18440.48,E2 -18440.48} C_VEL
LIN {X 0,Y 254.649,Z 605.487,A -85,B 0,C 180,E1 -18442.946,E2 -18442.946} C_VEL
LIN {X 0,Y 254.575,Z 610.098,A -85,B 0,C 180,E1 -18445.25,E2 -18445.25} C_VEL
LIN {X 0,Y 254.563,Z 613.716,A -85,B 0,C 180,E1 -18447.627,E2 -18447.627} C_VEL
LIN {X 0,Y 254.675,Z 616.257,A -85,B 0,C 180,E1 -18450,E2 -18450} C_VEL
LIN {X 0,Y 254.457,Z 617.349,A -85,B 0,C 180,E1 -18451.583,E2 -18451.583} C_VEL
LIN {X 0,Y 254.16,Z 618.359,A -85,B 0,C 180,E1 -18454.759,E2 -18454.759} C_VEL
LIN {X 0,Y 254.15,Z 618.278,A -85,B 0,C 180,E1 -18456.351,E2 -18456.351} C_VEL
LIN {X 0,Y 254.634,Z 616.942,A -85,B 0,C 180,E1 -18459.533,E2 -18459.533} C_VEL
LIN {X 0,Y 255.784,Z 614.14,A -85,B 0,C 180,E1 -18462.698,E2 -18462.698} C_VEL
LIN {X 0,Y 257.29,Z 611.058,A -85,B 0,C 180,E1 -18465.041,E2 -18465.041} C_VEL
LIN {X 0,Y 260.035,Z 605.581,A -85,B 0,C 180,E1 -18468.109,E2 -18468.109} C_VEL
LIN {X 0,Y 263.546,Z 598.429,A -85,B 0,C 180,E1 -18471.1,E2 -18471.1} C_VEL
LIN {X 0,Y 267.587,Z 590.583,A -85,B 0,C 180,E1 -18473.612,E2 -18473.612} C_VEL
LIN {X 0,Y 272.28,Z 581.099,A -85,B 0,C 180,E1 -18476.028,E2 -18476.028} C_VEL
LIN {X 0,Y 275.323,Z 573.345,A -85,B 0,C 180,E1 -18477.766,E2 -18477.766} C_VEL
LIN {X 0,Y 276.867,Z 566.899,A -85,B 0,C 180,E1 -18479.288,E2 -18479.288} C_VEL
LIN {X 0,Y 277.993,Z 557.408,A -85,B 0,C 180,E1 -18481.64,E2 -18481.64} C_VEL
LIN {X 0,Y 278.147,Z 548.471,A -85,B 0,C 180,E1 -18484.113,E2 -18484.113} C_VEL
LIN {X 0,Y 277.879,Z 541.589,A -85,B 0,C 180,E1 -18486.308,E2 -18486.308} C_VEL
LIN {X 0,Y 277.575,Z 537.471,A -85,B 0,C 180,E1 -18487.833,E2 -18487.833} C_VEL
LIN {X 0,Y 277.271,Z 534.039,A -85,B 0,C 180,E1 -18489.322,E2 -18489.322} C_VEL
LIN {X 0,Y 276.369,Z 529.513,A -85,B 0,C 180,E1 -18492.484,E2 -18492.484} C_VEL
LIN {X 0,Y 276.348,Z 528.37,A -85,B 0,C 180,E1 -18493.366,E2 -18493.366} C_VEL
LIN {X 0,Y 276.321,Z 526.888,A -85,B 0,C 180,E1 -18495.411,E2 -18495.411} C_VEL
LIN {X 0,Y 276.305,Z 526.873,A -85,B 0,C 180,E1 -18497.531,E2 -18497.531} C_VEL
LIN {X 0,Y 277.237,Z 528.115,A -85,B 0,C 180,E1 -18500.673,E2 -18500.673} C_VEL
LIN {X 0,Y 278.284,Z 529.718,A -85,B 0,C 180,E1 -18502.691,E2 -18502.691} C_VEL
LIN {X 0,Y 279.416,Z 532.253,A -85,B 0,C 180,E1 -18504.655,E2 -18504.655} C_VEL
LIN {X 0,Y 280.842,Z 536.947,A -85,B 0,C 180,E1 -18507.196,E2 -18507.196} C_VEL
LIN {X 0,Y 281.852,Z 541.841,A -85,B 0,C 180,E1 -18509.286,E2 -18509.286} C_VEL
LIN {X 0,Y 282.411,Z 547.604,A -85,B 0,C 180,E1 -18511.393,E2 -18511.393} C_VEL
LIN {X 0,Y 282.441,Z 548.786,A -85,B 0,C 180,E1 -18511.785,E2 -18511.785} C_VEL
LIN {X 0,Y 282.002,Z 550.429,A -85,B 0,C 180,E1 -18512.188,E2 -18512.188} C_VEL
LIN {X 0,Y 276.837,Z 560.993,A -85,B 0,C 180,E1 -18514.433,E2 -18514.433} C_VEL
LIN {X 0,Y 272.731,Z 568.589,A -85,B 0,C 180,E1 -18516.458,E2 -18516.458} C_VEL
LIN {X 0,Y 269.008,Z 574.895,A -85,B 0,C 180,E1 -18518.546,E2 -18518.546} C_VEL
LIN {X 0,Y 264.829,Z 581.623,A -85,B 0,C 180,E1 -18521.431,E2 -18521.431} C_VEL
LIN {X 0,Y 261.46,Z 586.535,A -85,B 0,C 180,E1 -18524.408,E2 -18524.408} C_VEL
LIN {X 0,Y 259.923,Z 588.446,A -85,B 0,C 180,E1 -18525.916,E2 -18525.916} C_VEL
LIN {X 0,Y 257.705,Z 591.022,A -85,B 0,C 180,E1 -18528.995,E2 -18528.995} C_VEL
LIN {X 0,Y 255.892,Z 592.147,A -85,B 0,C 180,E1 -18532.107,E2 -18532.107} C_VEL
LIN {X 0,Y 255.039,Z 591.768,A -85,B 0,C 180,E1 -18535.258,E2 -18535.258} C_VEL
LIN {X 0,Y 254.419,Z 589.833,A -85,B 0,C 180,E1 -18538.417,E2 -18538.417} C_VEL
LIN {X 0,Y 254.267,Z 586.343,A -85,B 0,C 180,E1 -18541.584,E2 -18541.584} C_VEL
LIN {X 0,Y 254.376,Z 582.588,A -85,B 0,C 180,E1 -18543.961,E2 -18543.961} C_VEL
LIN {X 0,Y 254.567,Z 577.765,A -85,B 0,C 180,E1 -18546.341,E2 -18546.341} C_VEL
LIN {X 0,Y 254.999,Z 571.706,A -85,B 0,C 180,E1 -18548.719,E2 -18548.719} C_VEL
LIN {X 0,Y 255.638,Z 564.24,A -85,B 0,C 180,E1 -18551.096,E2 -18551.096} C_VEL
LIN {X 0,Y 256.559,Z 555.146,A -85,B 0,C 180,E1 -18553.465,E2 -18553.465} C_VEL
LIN {X 0,Y 257.747,Z 544.935,A -85,B 0,C 180,E1 -18555.621,E2 -18555.621} C_VEL
LIN {X 0,Y 258.946,Z 534.883,A -85,B 0,C 180,E1 -18557.371,E2 -18557.371} C_VEL
LIN {X 0,Y 259.929,Z 524.084,A -85,B 0,C 180,E1 -18558.933,E2 -18558.933} C_VEL
LIN {X 0,Y 260.446,Z 517.737,A -85,B 0,C 180,E1 -18559.713,E2 -18559.713} C_VEL
LIN {X 0,Y 257.879,Z 503.904,A -85,B 0,C 180,E1 -18561.236,E2 -18561.236} C_VEL
LIN {X 0,Y 255.297,Z 489.755,A -85,B 0,C 180,E1 -18562.437,E2 -18562.437} C_VEL
LIN {X 0,Y 254.666,Z 485.724,A -85,B 0,C 180,E1 -18562.729,E2 -18562.729} C_VEL
LIN {X 0,Y 254.733,Z 484.762,A -85,B 0,C 180,E1 -18564.014,E2 -18564.014} C_VEL
LIN {X 0,Y 255.214,Z 484.697,A -85,B 0,C 180,E1 -18568.211,E2 -18568.211} C_VEL
LIN {X 0,Y 255.557,Z 484.648,A -85,B 0,C 180,E1 -18571.512,E2 -18571.512} C_VEL
LIN {X 0,Y 255.881,Z 484.608,A -85,B 0,C 180,E1 -18575.225,E2 -18575.225} C_VEL
LIN {X 0,Y 256.05,Z 484.587,A -85,B 0,C 180,E1 -18579.147,E2 -18579.147} C_VEL
LIN {X 0,Y 256.065,Z 484.585,A -85,B 0,C 180,E1 -18583.327,E2 -18583.327} C_VEL
LIN {X 0,Y 256.076,Z 484.586,A -85,B 0,C 180,E1 -18587.819,E2 -18587.819} C_VEL
LIN {X 0,Y 256.092,Z 484.581,A -85,B 0,C 180,E1 -18590.861,E2 -18590.861} C_VEL
LIN {X 0,Y 256.12,Z 484.58,A -85,B 0,C 180,E1 -18594.813,E2 -18594.813} C_VEL
LIN {X 0,Y 256.097,Z 484.581,A -85,B 0,C 180,E1 -18598.572,E2 -18598.572} C_VEL
LIN {X 0,Y 256.144,Z 484.581,A -85,B 0,C 180,E1 -18602.196,E2 -18602.196} C_VEL
LIN {X 0,Y 256.172,Z 484.574,A -85,B 0,C 180,E1 -18605.699,E2 -18605.699} C_VEL
LIN {X 0,Y 256.172,Z 484.571,A -85,B 0,C 180,E1 -18609.105,E2 -18609.105} C_VEL
LIN {X 0,Y 256.305,Z 484.56,A -85,B 0,C 180,E1 -18614.085,E2 -18614.085} C_VEL
LIN {X 0,Y 256.302,Z 484.556,A -85,B 0,C 180,E1 -18618.933,E2 -18618.933} C_VEL
LIN {X 0,Y 256.52,Z 484.533,A -85,B 0,C 180,E1 -18622.126,E2 -18622.126} C_VEL
LIN {X 0,Y 256.503,Z 484.53,A -85,B 0,C 180,E1 -18626.858,E2 -18626.858} C_VEL
LIN {X 0,Y 256.77,Z 484.503,A -85,B 0,C 180,E1 -18630,E2 -18630} C_VEL
LIN {X 0,Y 256.5,Z 484.531,A -85,B 0,C 180,E1 -18633.141,E2 -18633.141} C_VEL
LIN {X 0,Y 256.5,Z 484.535,A -85,B 0,C 180,E1 -18637.874,E2 -18637.874} C_VEL
LIN {X 0,Y 256.299,Z 484.555,A -85,B 0,C 180,E1 -18642.672,E2 -18642.672} C_VEL
LIN {X 0,Y 256.287,Z 484.56,A -85,B 0,C 180,E1 -18646.302,E2 -18646.302} C_VEL
LIN {X 0,Y 256.161,Z 484.573,A -85,B 0,C 180,E1 -18651.119,E2 -18651.119} C_VEL
LIN {X 0,Y 256.192,Z 484.57,A -85,B 0,C 180,E1 -18655.138,E2 -18655.138} C_VEL
LIN {X 0,Y 256.114,Z 484.582,A -85,B 0,C 180,E1 -18659.599,E2 -18659.599} C_VEL
LIN {X 0,Y 256.088,Z 484.584,A -85,B 0,C 180,E1 -18663.289,E2 -18663.289} C_VEL
LIN {X 0,Y 256.131,Z 484.579,A -85,B 0,C 180,E1 -18667.274,E2 -18667.274} C_VEL
LIN {X 0,Y 256.058,Z 484.586,A -85,B 0,C 180,E1 -18671.202,E2 -18671.202} C_VEL
LIN {X 0,Y 256.059,Z 484.59,A -85,B 0,C 180,E1 -18675.53,E2 -18675.53} C_VEL
LIN {X 0,Y 256.056,Z 484.585,A -85,B 0,C 180,E1 -18678.796,E2 -18678.796} C_VEL
LIN {X 0,Y 256.134,Z 484.578,A -85,B 0,C 180,E1 -18682.867,E2 -18682.867} C_VEL
LIN {X 0,Y 256.078,Z 484.582,A -85,B 0,C 180,E1 -18686.708,E2 -18686.708} C_VEL
LIN {X 0,Y 256.14,Z 484.579,A -85,B 0,C 180,E1 -18691.404,E2 -18691.404} C_VEL
LIN {X 0,Y 256.168,Z 484.575,A -85,B 0,C 180,E1 -18695.699,E2 -18695.699} C_VEL
LIN {X 0,Y 256.168,Z 484.574,A -85,B 0,C 180,E1 -18699.104,E2 -18699.104} C_VEL
LIN {X 0,Y 256.301,Z 484.555,A -85,B 0,C 180,E1 -18704.085,E2 -18704.085} C_VEL
LIN {X 0,Y 256.31,Z 484.556,A -85,B 0,C 180,E1 -18708.934,E2 -18708.934} C_VEL
LIN {X 0,Y 256.541,Z 484.526,A -85,B 0,C 180,E1 -18712.127,E2 -18712.127} C_VEL
LIN {X 0,Y 256.715,Z 484.505,A -85,B 0,C 180,E1 -18718.431,E2 -18718.431} C_VEL
LIN {X 0,Y 256.715,Z 484.507,A -85,B 0,C 180,E1 -18721.568,E2 -18721.568} C_VEL
LIN {X 0,Y 256.541,Z 484.528,A -85,B 0,C 180,E1 -18727.873,E2 -18727.873} C_VEL
LIN {X 0,Y 256.31,Z 484.555,A -85,B 0,C 180,E1 -18731.066,E2 -18731.066} C_VEL
LIN {X 0,Y 256.3,Z 484.558,A -85,B 0,C 180,E1 -18735.915,E2 -18735.915} C_VEL
LIN {X 0,Y 256.167,Z 484.573,A -85,B 0,C 180,E1 -18740.895,E2 -18740.895} C_VEL
LIN {X 0,Y 256.188,Z 484.574,A -85,B 0,C 180,E1 -18745.138,E2 -18745.138} C_VEL
LIN {X 0,Y 256.103,Z 484.583,A -85,B 0,C 180,E1 -18749.601,E2 -18749.601} C_VEL
LIN {X 0,Y 256.085,Z 484.588,A -85,B 0,C 180,E1 -18753.29,E2 -18753.29} C_VEL
LIN {X 0,Y 256.14,Z 484.579,A -85,B 0,C 180,E1 -18757.278,E2 -18757.278} C_VEL
LIN {X 0,Y 256.194,Z 484.57,A -85,B 0,C 180,E1 -18762.197,E2 -18762.197} C_VEL
LIN {X 0,Y 255.973,Z 484.849,A -85,B 0,C 180,E1 -18763.073,E2 -18763.073} C_VEL
LIN {X 0,Y 255.278,Z 485.572,A -85,B 0,C 180,E1 -18763.929,E2 -18763.929} C_VEL
LIN {X 0,Y 251.073,Z 489.938,A -85,B 0,C 180,E1 -18767.282,E2 -18767.282} C_VEL
LIN {X 0,Y 250.352,Z 491.553,A -85,B 0,C 180,E1 -18768.584,E2 -18768.584} C_VEL
LIN {X 0,Y 250.388,Z 492.074,A -85,B 0,C 180,E1 -18769.023,E2 -18769.023} C_VEL
LIN {X 0,Y 250.988,Z 495.612,A -85,B 0,C 180,E1 -18771.974,E2 -18771.974} C_VEL
LIN {X 0,Y 250.949,Z 498.502,A -85,B 0,C 180,E1 -18774.308,E2 -18774.308} C_VEL
LIN {X 0,Y 250.045,Z 502.874,A -85,B 0,C 180,E1 -18777.722,E2 -18777.722} C_VEL
LIN {X 0,Y 248.972,Z 508.701,A -85,B 0,C 180,E1 -18782.241,E2 -18782.241} C_VEL
LIN {X 0,Y 248.078,Z 514.888,A -85,B 0,C 180,E1 -18786.876,E2 -18786.876} C_VEL
LIN {X 0,Y 248.834,Z 527.235,A -85,B 0,C 180,E1 -18787.782,E2 -18787.782} C_VEL
LIN {X 0,Y 250.033,Z 540.863,A -85,B 0,C 180,E1 -18789.107,E2 -18789.107} C_VEL
LIN {X 0,Y 251.188,Z 553.093,A -85,B 0,C 180,E1 -18790.608,E2 -18790.608} C_VEL
LIN {X 0,Y 251.743,Z 560.353,A -85,B 0,C 180,E1 -18791.657,E2 -18791.657} C_VEL
LIN {X 0,Y 250.392,Z 572.247,A -85,B 0,C 180,E1 -18793.7,E2 -18793.7} C_VEL
LIN {X 0,Y 249.348,Z 581.768,A -85,B 0,C 180,E1 -18795.723,E2 -18795.723} C_VEL
LIN {X 0,Y 248.441,Z 591.122,A -85,B 0,C 180,E1 -18798.166,E2 -18798.166} C_VEL
LIN {X 0,Y 247.897,Z 598.723,A -85,B 0,C 180,E1 -18800.618,E2 -18800.618} C_VEL
LIN {X 0,Y 247.634,Z 603.879,A -85,B 0,C 180,E1 -18802.663,E2 -18802.663} C_VEL
LIN {X 0,Y 247.53,Z 608.852,A -85,B 0,C 180,E1 -18805.114,E2 -18805.114} C_VEL
LIN {X 0,Y 247.522,Z 612.627,A -85,B 0,C 180,E1 -18807.559,E2 -18807.559} C_VEL
LIN {X 0,Y 247.64,Z 615.335,A -85,B 0,C 180,E1 -18810,E2 -18810} C_VEL
LIN {X 0,Y 247.412,Z 616.559,A -85,B 0,C 180,E1 -18811.628,E2 -18811.628} C_VEL
LIN {X 0,Y 247.081,Z 617.744,A -85,B 0,C 180,E1 -18814.896,E2 -18814.896} C_VEL
LIN {X 0,Y 247.25,Z 617.429,A -85,B 0,C 180,E1 -18818.171,E2 -18818.171} C_VEL
LIN {X 0,Y 248.136,Z 615.62,A -85,B 0,C 180,E1 -18821.436,E2 -18821.436} C_VEL
LIN {X 0,Y 249.814,Z 612.349,A -85,B 0,C 180,E1 -18824.667,E2 -18824.667} C_VEL
LIN {X 0,Y 252.564,Z 607.599,A -85,B 0,C 180,E1 -18827.824,E2 -18827.824} C_VEL
LIN {X 0,Y 255.38,Z 602.325,A -85,B 0,C 180,E1 -18830.461,E2 -18830.461} C_VEL
LIN {X 0,Y 259.325,Z 595.352,A -85,B 0,C 180,E1 -18833.14,E2 -18833.14} C_VEL
LIN {X 0,Y 263.903,Z 587.081,A -85,B 0,C 180,E1 -18835.643,E2 -18835.643} C_VEL
LIN {X 0,Y 268.201,Z 578.726,A -85,B 0,C 180,E1 -18837.719,E2 -18837.719} C_VEL
LIN {X 0,Y 270.387,Z 572.726,A -85,B 0,C 180,E1 -18839.167,E2 -18839.167} C_VEL
LIN {X 0,Y 272.018,Z 565.265,A -85,B 0,C 180,E1 -18841.114,E2 -18841.114} C_VEL
LIN {X 0,Y 272.926,Z 557.855,A -85,B 0,C 180,E1 -18843.151,E2 -18843.151} C_VEL
LIN {X 0,Y 273.332,Z 550.447,A -85,B 0,C 180,E1 -18845.438,E2 -18845.438} C_VEL
LIN {X 0,Y 273.396,Z 543.162,A -85,B 0,C 180,E1 -18848.094,E2 -18848.094} C_VEL
LIN {X 0,Y 273.168,Z 539.137,A -85,B 0,C 180,E1 -18850.031,E2 -18850.031} C_VEL
LIN {X 0,Y 272.742,Z 534.191,A -85,B 0,C 180,E1 -18853.822,E2 -18853.822} C_VEL
LIN {X 0,Y 272.761,Z 532.956,A -85,B 0,C 180,E1 -18856.175,E2 -18856.175} C_VEL
LIN {X 0,Y 272.832,Z 533.263,A -85,B 0,C 180,E1 -18858.334,E2 -18858.334} C_VEL
LIN {X 0,Y 273.423,Z 534.054,A -85,B 0,C 180,E1 -18860.455,E2 -18860.455} C_VEL
LIN {X 0,Y 274.346,Z 535.614,A -85,B 0,C 180,E1 -18862.575,E2 -18862.575} C_VEL
LIN {X 0,Y 275.326,Z 538.378,A -85,B 0,C 180,E1 -18864.77,E2 -18864.77} C_VEL
LIN {X 0,Y 276.551,Z 543.816,A -85,B 0,C 180,E1 -18867.746,E2 -18867.746} C_VEL
LIN {X 0,Y 277.029,Z 549.831,A -85,B 0,C 180,E1 -18870.257,E2 -18870.257} C_VEL
LIN {X 0,Y 276.967,Z 552.275,A -85,B 0,C 180,E1 -18871.176,E2 -18871.176} C_VEL
LIN {X 0,Y 272.389,Z 561.263,A -85,B 0,C 180,E1 -18873.159,E2 -18873.159} C_VEL
LIN {X 0,Y 267.248,Z 569.952,A -85,B 0,C 180,E1 -18875.532,E2 -18875.532} C_VEL
LIN {X 0,Y 262.692,Z 577.046,A -85,B 0,C 180,E1 -18878.004,E2 -18878.004} C_VEL
LIN {X 0,Y 258.294,Z 583.292,A -85,B 0,C 180,E1 -18880.943,E2 -18880.943} C_VEL
LIN {X 0,Y 254.756,Z 587.903,A -85,B 0,C 180,E1 -18883.986,E2 -18883.986} C_VEL
LIN {X 0,Y 253.143,Z 589.607,A -85,B 0,C 180,E1 -18885.531,E2 -18885.531} C_VEL
LIN {X 0,Y 250.684,Z 591.997,A -85,B 0,C 180,E1 -18888.885,E2 -18888.885} C_VEL
LIN {X 0,Y 248.909,Z 592.762,A -85,B 0,C 180,E1 -18891.884,E2 -18891.884} C_VEL
LIN {X 0,Y 247.983,Z 592.081,A -85,B 0,C 180,E1 -18895.123,E2 -18895.123} C_VEL
LIN {X 0,Y 247.341,Z 589.933,A -85,B 0,C 180,E1 -18898.372,E2 -18898.372} C_VEL
LIN {X 0,Y 247.173,Z 587.269,A -85,B 0,C 180,E1 -18900.815,E2 -18900.815} C_VEL
LIN {X 0,Y 247.244,Z 583.638,A -85,B 0,C 180,E1 -18903.259,E2 -18903.259} C_VEL
LIN {X 0,Y 247.347,Z 579.411,A -85,B 0,C 180,E1 -18905.49,E2 -18905.49} C_VEL
LIN {X 0,Y 247.833,Z 573.131,A -85,B 0,C 180,E1 -18908.152,E2 -18908.152} C_VEL
LIN {X 0,Y 248.42,Z 565.958,A -85,B 0,C 180,E1 -18910.597,E2 -18910.597} C_VEL
LIN {X 0,Y 249.298,Z 557.139,A -85,B 0,C 180,E1 -18913.034,E2 -18913.034} C_VEL
LIN {X 0,Y 250.272,Z 548.263,A -85,B 0,C 180,E1 -18915.056,E2 -18915.056} C_VEL
LIN {X 0,Y 251.476,Z 537.592,A -85,B 0,C 180,E1 -18917.065,E2 -18917.065} C_VEL
LIN {X 0,Y 252.545,Z 527.02,A -85,B 0,C 180,E1 -18918.698,E2 -18918.698} C_VEL
LIN {X 0,Y 253.282,Z 517.991,A -85,B 0,C 180,E1 -18919.872,E2 -18919.872} C_VEL
LIN {X 0,Y 250.861,Z 504.935,A -85,B 0,C 180,E1 -18921.359,E2 -18921.359} C_VEL
LIN {X 0,Y 248.302,Z 490.729,A -85,B 0,C 180,E1 -18922.622,E2 -18922.622} C_VEL
LIN {X 0,Y 247.61,Z 486.118,A -85,B 0,C 180,E1 -18922.972,E2 -18922.972} C_VEL
LIN {X 0,Y 247.66,Z 485.641,A -85,B 0,C 180,E1 -18923.808,E2 -18923.808} C_VEL
LIN {X 0,Y 248.192,Z 485.569,A -85,B 0,C 180,E1 -18928.618,E2 -18928.618} C_VEL
LIN {X 0,Y 248.57,Z 485.52,A -85,B 0,C 180,E1 -18932.494,E2 -18932.494} C_VEL
LIN {X 0,Y 248.886,Z 485.484,A -85,B 0,C 180,E1 -18936.371,E2 -18936.371} C_VEL
LIN {X 0,Y 248.992,Z 485.469,A -85,B 0,C 180,E1 -18940.35,E2 -18940.35} C_VEL
LIN {X 0,Y 249.013,Z 485.464,A -85,B 0,C 180,E1 -18942.793,E2 -18942.793} C_VEL
LIN {X 0,Y 249.02,Z 485.464,A -85,B 0,C 180,E1 -18947.363,E2 -18947.363} C_VEL
LIN {X 0,Y 249.041,Z 485.46,A -85,B 0,C 180,E1 -18951.621,E2 -18951.621} C_VEL
LIN {X 0,Y 249.063,Z 485.459,A -85,B 0,C 180,E1 -18955.642,E2 -18955.642} C_VEL
LIN {X 0,Y 249.055,Z 485.457,A -85,B 0,C 180,E1 -18959.473,E2 -18959.473} C_VEL
LIN {X 0,Y 249.077,Z 485.457,A -85,B 0,C 180,E1 -18963.162,E2 -18963.162} C_VEL
LIN {X 0,Y 249.084,Z 485.455,A -85,B 0,C 180,E1 -18966.733,E2 -18966.733} C_VEL
LIN {X 0,Y 249.116,Z 485.455,A -85,B 0,C 180,E1 -18970.212,E2 -18970.212} C_VEL
LIN {X 0,Y 249.247,Z 485.437,A -85,B 0,C 180,E1 -18973.622,E2 -18973.622} C_VEL
LIN {X 0,Y 249.25,Z 485.435,A -85,B 0,C 180,E1 -18978.616,E2 -18978.616} C_VEL
LIN {X 0,Y 249.459,Z 485.412,A -85,B 0,C 180,E1 -18981.902,E2 -18981.902} C_VEL
LIN {X 0,Y 249.3,Z 485.427,A -85,B 0,C 180,E1 -18985.148,E2 -18985.148} C_VEL
LIN {X 0,Y 249.68,Z 485.383,A -85,B 0,C 180,E1 -18988.387,E2 -18988.387} C_VEL
LIN {X 0,Y 249.68,Z 485.383,A -85,B 0,C 180,E1 -18991.613,E2 -18991.613} C_VEL
LIN {X 0,Y 249.442,Z 485.412,A -85,B 0,C 180,E1 -18996.471,E2 -18996.471} C_VEL
LIN {X 0,Y 249.348,Z 485.426,A -85,B 0,C 180,E1 -18999.736,E2 -18999.736} C_VEL
LIN {X 0,Y 249.21,Z 485.439,A -85,B 0,C 180,E1 -19004.703,E2 -19004.703} C_VEL
LIN {X 0,Y 249.144,Z 485.451,A -85,B 0,C 180,E1 -19008.077,E2 -19008.077} C_VEL
LIN {X 0,Y 249.091,Z 485.455,A -85,B 0,C 180,E1 -19011.517,E2 -19011.517} C_VEL
LIN {X 0,Y 249.134,Z 485.451,A -85,B 0,C 180,E1 -19015.482,E2 -19015.482} C_VEL
LIN {X 0,Y 249.083,Z 485.455,A -85,B 0,C 180,E1 -19018.991,E2 -19018.991} C_VEL
LIN {X 0,Y 249.039,Z 485.461,A -85,B 0,C 180,E1 -19022.424,E2 -19022.424} C_VEL
LIN {X 0,Y 249.072,Z 485.458,A -85,B 0,C 180,E1 -19026.338,E2 -19026.338} C_VEL
LIN {X 0,Y 249.028,Z 485.462,A -85,B 0,C 180,E1 -19030.473,E2 -19030.473} C_VEL
LIN {X 0,Y 249.004,Z 485.466,A -85,B 0,C 180,E1 -19034.879,E2 -19034.879} C_VEL
LIN {X 0,Y 249.018,Z 485.465,A -85,B 0,C 180,E1 -19037.362,E2 -19037.362} C_VEL
LIN {X 0,Y 249.046,Z 485.462,A -85,B 0,C 180,E1 -19042.199,E2 -19042.199} C_VEL
LIN {X 0,Y 249.058,Z 485.462,A -85,B 0,C 180,E1 -19045.641,E2 -19045.641} C_VEL
LIN {X 0,Y 249.053,Z 485.461,A -85,B 0,C 180,E1 -19049.473,E2 -19049.473} C_VEL
LIN {X 0,Y 249.075,Z 485.458,A -85,B 0,C 180,E1 -19053.162,E2 -19053.162} C_VEL
LIN {X 0,Y 249.08,Z 485.454,A -85,B 0,C 180,E1 -19056.732,E2 -19056.732} C_VEL
LIN {X 0,Y 249.112,Z 485.453,A -85,B 0,C 180,E1 -19060.211,E2 -19060.211} C_VEL
LIN {X 0,Y 249.243,Z 485.437,A -85,B 0,C 180,E1 -19063.621,E2 -19063.621} C_VEL
LIN {X 0,Y 249.254,Z 485.435,A -85,B 0,C 180,E1 -19068.616,E2 -19068.616} C_VEL
LIN {X 0,Y 249.485,Z 485.406,A -85,B 0,C 180,E1 -19071.903,E2 -19071.903} C_VEL
LIN {X 0,Y 249.438,Z 485.412,A -85,B 0,C 180,E1 -19076.769,E2 -19076.769} C_VEL
LIN {X 0,Y 249.729,Z 485.375,A -85,B 0,C 180,E1 -19080,E2 -19080} C_VEL
LIN {X 0,Y 249.436,Z 485.412,A -85,B 0,C 180,E1 -19083.23,E2 -19083.23} C_VEL
LIN {X 0,Y 249.485,Z 485.406,A -85,B 0,C 180,E1 -19088.097,E2 -19088.097} C_VEL
LIN {X 0,Y 249.253,Z 485.436,A -85,B 0,C 180,E1 -19091.383,E2 -19091.383} C_VEL
LIN {X 0,Y 249.242,Z 485.436,A -85,B 0,C 180,E1 -19096.378,E2 -19096.378} C_VEL
LIN {X 0,Y 249.087,Z 485.458,A -85,B 0,C 180,E1 -19101.518,E2 -19101.518} C_VEL
LIN {X 0,Y 249.13,Z 485.453,A -85,B 0,C 180,E1 -19105.482,E2 -19105.482} C_VEL
LIN {X 0,Y 249.072,Z 485.456,A -85,B 0,C 180,E1 -19108.989,E2 -19108.989} C_VEL
LIN {X 0,Y 249.035,Z 485.462,A -85,B 0,C 180,E1 -19112.425,E2 -19112.425} C_VEL
LIN {X 0,Y 249.074,Z 485.455,A -85,B 0,C 180,E1 -19116.338,E2 -19116.338} C_VEL
LIN {X 0,Y 249.084,Z 485.456,A -85,B 0,C 180,E1 -19120.462,E2 -19120.462} C_VEL
LIN {X 0,Y 249.238,Z 485.579,A -85,B 0,C 180,E1 -19123.349,E2 -19123.349} C_VEL
LIN {X 0,Y 250.07,Z 490.39,A -85,B 0,C 180,E1 -19127.585,E2 -19127.585} C_VEL
LIN {X 0,Y 250.388,Z 492.074,A -85,B 0,C 180,E1 -19129.023,E2 -19129.023} C_VEL
LIN {X 0,Y 250.032,Z 493.675,A -85,B 0,C 180,E1 -19130.321,E2 -19130.321} C_VEL
LIN {X 0,Y 248.651,Z 495.344,A -85,B 0,C 180,E1 -19131.594,E2 -19131.594} C_VEL
LIN {X 0,Y 243.979,Z 499.867,A -85,B 0,C 180,E1 -19135.023,E2 -19135.023} C_VEL
LIN {X 0,Y 243.444,Z 501,A -85,B 0,C 180,E1 -19135.924,E2 -19135.924} C_VEL
LIN {X 0,Y 242.24,Z 506.696,A -85,B 0,C 180,E1 -19140.502,E2 -19140.502} C_VEL
LIN {X 0,Y 241.395,Z 511.686,A -85,B 0,C 180,E1 -19144.493,E2 -19144.493} C_VEL
LIN {X 0,Y 241.016,Z 514.308,A -85,B 0,C 180,E1 -19146.591,E2 -19146.591} C_VEL
LIN {X 0,Y 241.945,Z 529.557,A -85,B 0,C 180,E1 -19147.814,E2 -19147.814} C_VEL
LIN {X 0,Y 243.107,Z 543.519,A -85,B 0,C 180,E1 -19149.295,E2 -19149.295} C_VEL
LIN {X 0,Y 244.327,Z 555.55,A -85,B 0,C 180,E1 -19150.902,E2 -19150.902} C_VEL
LIN {X 0,Y 244.582,Z 560.716,A -85,B 0,C 180,E1 -19151.697,E2 -19151.697} C_VEL
LIN {X 0,Y 243.318,Z 571.661,A -85,B 0,C 180,E1 -19153.644,E2 -19153.644} C_VEL
LIN {X 0,Y 242.292,Z 581.214,A -85,B 0,C 180,E1 -19155.727,E2 -19155.727} C_VEL
LIN {X 0,Y 241.378,Z 590.55,A -85,B 0,C 180,E1 -19158.24,E2 -19158.24} C_VEL
LIN {X 0,Y 240.86,Z 598.115,A -85,B 0,C 180,E1 -19160.765,E2 -19160.765} C_VEL
LIN {X 0,Y 240.575,Z 604.263,A -85,B 0,C 180,E1 -19163.341,E2 -19163.341} C_VEL
LIN {X 0,Y 240.523,Z 608.932,A -85,B 0,C 180,E1 -19165.811,E2 -19165.811} C_VEL
LIN {X 0,Y 240.568,Z 612.553,A -85,B 0,C 180,E1 -19168.326,E2 -19168.326} C_VEL
LIN {X 0,Y 240.625,Z 614.358,A -85,B 0,C 180,E1 -19170,E2 -19170} C_VEL
LIN {X 0,Y 240.364,Z 615.675,A -85,B 0,C 180,E1 -19171.676,E2 -19171.676} C_VEL
LIN {X 0,Y 240.011,Z 617.117,A -85,B 0,C 180,E1 -19175.04,E2 -19175.04} C_VEL
LIN {X 0,Y 240.2,Z 617.01,A -85,B 0,C 180,E1 -19178.413,E2 -19178.413} C_VEL
LIN {X 0,Y 241.16,Z 615.471,A -85,B 0,C 180,E1 -19181.771,E2 -19181.771} C_VEL
LIN {X 0,Y 242.962,Z 612.508,A -85,B 0,C 180,E1 -19185.09,E2 -19185.09} C_VEL
LIN {X 0,Y 245.823,Z 608.06,A -85,B 0,C 180,E1 -19188.33,E2 -19188.33} C_VEL
LIN {X 0,Y 249.391,Z 602.129,A -85,B 0,C 180,E1 -19191.491,E2 -19191.491} C_VEL
LIN {X 0,Y 253.579,Z 595.533,A -85,B 0,C 180,E1 -19194.13,E2 -19194.13} C_VEL
LIN {X 0,Y 259.174,Z 586.259,A -85,B 0,C 180,E1 -19197.015,E2 -19197.015} C_VEL
LIN {X 0,Y 262.835,Z 579.429,A -85,B 0,C 180,E1 -19198.771,E2 -19198.771} C_VEL
LIN {X 0,Y 265.071,Z 573.826,A -85,B 0,C 180,E1 -19200.249,E2 -19200.249} C_VEL
LIN {X 0,Y 267.129,Z 565.283,A -85,B 0,C 180,E1 -19202.659,E2 -19202.659} C_VEL
LIN {X 0,Y 268.237,Z 557.201,A -85,B 0,C 180,E1 -19205.199,E2 -19205.199} C_VEL
LIN {X 0,Y 268.761,Z 551.027,A -85,B 0,C 180,E1 -19207.42,E2 -19207.42} C_VEL
LIN {X 0,Y 269.004,Z 546.074,A -85,B 0,C 180,E1 -19209.583,E2 -19209.583} C_VEL
LIN {X 0,Y 268.79,Z 542.948,A -85,B 0,C 180,E1 -19211.628,E2 -19211.628} C_VEL
LIN {X 0,Y 268.804,Z 541.325,A -85,B 0,C 180,E1 -19212.94,E2 -19212.94} C_VEL
LIN {X 0,Y 268.907,Z 539.443,A -85,B 0,C 180,E1 -19215.117,E2 -19215.117} C_VEL
LIN {X 0,Y 268.933,Z 539.036,A -85,B 0,C 180,E1 -19217.199,E2 -19217.199} C_VEL
LIN {X 0,Y 269.115,Z 539.526,A -85,B 0,C 180,E1 -19219.241,E2 -19219.241} C_VEL
LIN {X 0,Y 269.786,Z 540.534,A -85,B 0,C 180,E1 -19221.4,E2 -19221.4} C_VEL
LIN {X 0,Y 270.571,Z 542.623,A -85,B 0,C 180,E1 -19223.632,E2 -19223.632} C_VEL
LIN {X 0,Y 271.258,Z 546.123,A -85,B 0,C 180,E1 -19226.006,E2 -19226.006} C_VEL
LIN {X 0,Y 271.696,Z 550.367,A -85,B 0,C 180,E1 -19228.221,E2 -19228.221} C_VEL
LIN {X 0,Y 271.657,Z 554.676,A -85,B 0,C 180,E1 -19230.085,E2 -19230.085} C_VEL
LIN {X 0,Y 271.437,Z 555.914,A -85,B 0,C 180,E1 -19230.532,E2 -19230.532} C_VEL
LIN {X 0,Y 265.683,Z 565.616,A -85,B 0,C 180,E1 -19232.851,E2 -19232.851} C_VEL
LIN {X 0,Y 260.459,Z 573.55,A -85,B 0,C 180,E1 -19235.277,E2 -19235.277} C_VEL
LIN {X 0,Y 256.386,Z 579.126,A -85,B 0,C 180,E1 -19237.433,E2 -19237.433} C_VEL
LIN {X 0,Y 251.795,Z 585.002,A -85,B 0,C 180,E1 -19240.431,E2 -19240.431} C_VEL
LIN {X 0,Y 248.055,Z 589.202,A -85,B 0,C 180,E1 -19243.542,E2 -19243.542} C_VEL
LIN {X 0,Y 246.381,Z 590.768,A -85,B 0,C 180,E1 -19245.125,E2 -19245.125} C_VEL
LIN {X 0,Y 243.922,Z 592.752,A -85,B 0,C 180,E1 -19248.365,E2 -19248.365} C_VEL
LIN {X 0,Y 241.908,Z 593.3,A -85,B 0,C 180,E1 -19251.648,E2 -19251.648} C_VEL
LIN {X 0,Y 240.931,Z 592.38,A -85,B 0,C 180,E1 -19254.98,E2 -19254.98} C_VEL
LIN {X 0,Y 240.54,Z 591.367,A -85,B 0,C 180,E1 -19256.65,E2 -19256.65} C_VEL
LIN {X 0,Y 240.125,Z 588.134,A -85,B 0,C 180,E1 -19260,E2 -19260} C_VEL
LIN {X 0,Y 240.157,Z 584.651,A -85,B 0,C 180,E1 -19262.516,E2 -19262.516} C_VEL
LIN {X 0,Y 240.241,Z 579.451,A -85,B 0,C 180,E1 -19265.375,E2 -19265.375} C_VEL
LIN {X 0,Y 240.719,Z 573.373,A -85,B 0,C 180,E1 -19267.989,E2 -19267.989} C_VEL
LIN {X 0,Y 241.285,Z 566.179,A -85,B 0,C 180,E1 -19270.489,E2 -19270.489} C_VEL
LIN {X 0,Y 242.167,Z 557.345,A -85,B 0,C 180,E1 -19272.998,E2 -19272.998} C_VEL
LIN {X 0,Y 243.136,Z 548.504,A -85,B 0,C 180,E1 -19275.079,E2 -19275.079} C_VEL
LIN {X 0,Y 244.357,Z 537.889,A -85,B 0,C 180,E1 -19277.146,E2 -19277.146} C_VEL
LIN {X 0,Y 245.274,Z 528.915,A -85,B 0,C 180,E1 -19278.598,E2 -19278.598} C_VEL
LIN {X 0,Y 246.242,Z 519.489,A -85,B 0,C 180,E1 -19279.884,E2 -19279.884} C_VEL
LIN {X 0,Y 243.946,Z 506.53,A -85,B 0,C 180,E1 -19281.428,E2 -19281.428} C_VEL
LIN {X 0,Y 241.476,Z 492.645,A -85,B 0,C 180,E1 -19282.743,E2 -19282.743} C_VEL
LIN {X 0,Y 240.545,Z 486.525,A -85,B 0,C 180,E1 -19283.231,E2 -19283.231} C_VEL
LIN {X 0,Y 241.031,Z 486.464,A -85,B 0,C 180,E1 -19287.81,E2 -19287.81} C_VEL
LIN {X 0,Y 241.52,Z 486.399,A -85,B 0,C 180,E1 -19292.448,E2 -19292.448} C_VEL
LIN {X 0,Y 241.794,Z 486.363,A -85,B 0,C 180,E1 -19295.544,E2 -19295.544} C_VEL
LIN {X 0,Y 241.953,Z 486.347,A -85,B 0,C 180,E1 -19298.346,E2 -19298.346} C_VEL
LIN {X 0,Y 241.937,Z 486.345,A -85,B 0,C 180,E1 -19301.923,E2 -19301.923} C_VEL
LIN {X 0,Y 241.938,Z 486.348,A -85,B 0,C 180,E1 -19306.571,E2 -19306.571} C_VEL
LIN {X 0,Y 241.976,Z 486.342,A -85,B 0,C 180,E1 -19310.284,E2 -19310.284} C_VEL
LIN {X 0,Y 242.041,Z 486.335,A -85,B 0,C 180,E1 -19314.498,E2 -19314.498} C_VEL
LIN {X 0,Y 241.979,Z 486.34,A -85,B 0,C 180,E1 -19318.48,E2 -19318.48} C_VEL
LIN {X 0,Y 242.011,Z 486.34,A -85,B 0,C 180,E1 -19322.313,E2 -19322.313} C_VEL
LIN {X 0,Y 242.062,Z 486.334,A -85,B 0,C 180,E1 -19326.016,E2 -19326.016} C_VEL
LIN {X 0,Y 242.043,Z 486.332,A -85,B 0,C 180,E1 -19329.608,E2 -19329.608} C_VEL
LIN {X 0,Y 242.168,Z 486.317,A -85,B 0,C 180,E1 -19333.278,E2 -19333.278} C_VEL
LIN {X 0,Y 242.186,Z 486.317,A -85,B 0,C 180,E1 -19338.279,E2 -19338.279} C_VEL
LIN {X 0,Y 242.405,Z 486.29,A -85,B 0,C 180,E1 -19341.664,E2 -19341.664} C_VEL
LIN {X 0,Y 242.261,Z 486.303,A -85,B 0,C 180,E1 -19345.007,E2 -19345.007} C_VEL
LIN {X 0,Y 242.641,Z 486.26,A -85,B 0,C 180,E1 -19348.34,E2 -19348.34} C_VEL
LIN {X 0,Y 242.641,Z 486.26,A -85,B 0,C 180,E1 -19351.659,E2 -19351.659} C_VEL
LIN {X 0,Y 242.413,Z 486.287,A -85,B 0,C 180,E1 -19356.659,E2 -19356.659} C_VEL
LIN {X 0,Y 242.272,Z 486.307,A -85,B 0,C 180,E1 -19360.023,E2 -19360.023} C_VEL
LIN {X 0,Y 242.171,Z 486.316,A -85,B 0,C 180,E1 -19365.14,E2 -19365.14} C_VEL
LIN {X 0,Y 242.077,Z 486.329,A -85,B 0,C 180,E1 -19368.623,E2 -19368.623} C_VEL
LIN {X 0,Y 242.017,Z 486.336,A -85,B 0,C 180,E1 -19372.179,E2 -19372.179} C_VEL
LIN {X 0,Y 242.07,Z 486.334,A -85,B 0,C 180,E1 -19375.837,E2 -19375.837} C_VEL
LIN {X 0,Y 242.032,Z 486.336,A -85,B 0,C 180,E1 -19379.58,E2 -19379.58} C_VEL
LIN {X 0,Y 241.994,Z 486.34,A -85,B 0,C 180,E1 -19383.49,E2 -19383.49} C_VEL
LIN {X 0,Y 242.005,Z 486.34,A -85,B 0,C 180,E1 -19387.579,E2 -19387.579} C_VEL
LIN {X 0,Y 241.945,Z 486.348,A -85,B 0,C 180,E1 -19391.92,E2 -19391.92} C_VEL
LIN {X 0,Y 241.936,Z 486.345,A -85,B 0,C 180,E1 -19396.571,E2 -19396.571} C_VEL
LIN {X 0,Y 241.958,Z 486.344,A -85,B 0,C 180,E1 -19400.28,E2 -19400.28} C_VEL
LIN {X 0,Y 242.006,Z 486.337,A -85,B 0,C 180,E1 -19404.492,E2 -19404.492} C_VEL
LIN {X 0,Y 241.977,Z 486.34,A -85,B 0,C 180,E1 -19408.479,E2 -19408.479} C_VEL
LIN {X 0,Y 242.01,Z 486.337,A -85,B 0,C 180,E1 -19412.312,E2 -19412.312} C_VEL
LIN {X 0,Y 242.058,Z 486.33,A -85,B 0,C 180,E1 -19416.015,E2 -19416.015} C_VEL
LIN {X 0,Y 242.039,Z 486.337,A -85,B 0,C 180,E1 -19419.608,E2 -19419.608} C_VEL
LIN {X 0,Y 242.164,Z 486.319,A -85,B 0,C 180,E1 -19423.278,E2 -19423.278} C_VEL
LIN {X 0,Y 242.187,Z 486.315,A -85,B 0,C 180,E1 -19428.279,E2 -19428.279} C_VEL
LIN {X 0,Y 242.436,Z 486.285,A -85,B 0,C 180,E1 -19431.665,E2 -19431.665} C_VEL
LIN {X 0,Y 242.262,Z 486.305,A -85,B 0,C 180,E1 -19435.007,E2 -19435.007} C_VEL
LIN {X 0,Y 242.638,Z 486.259,A -85,B 0,C 180,E1 -19438.34,E2 -19438.34} C_VEL
LIN {X 0,Y 242.637,Z 486.259,A -85,B 0,C 180,E1 -19441.659,E2 -19441.659} C_VEL
LIN {X 0,Y 242.434,Z 486.284,A -85,B 0,C 180,E1 -19446.658,E2 -19446.658} C_VEL
LIN {X 0,Y 242.346,Z 486.293,A -85,B 0,C 180,E1 -19450.02,E2 -19450.02} C_VEL
LIN {X 0,Y 242.167,Z 486.32,A -85,B 0,C 180,E1 -19455.14,E2 -19455.14} C_VEL
LIN {X 0,Y 242.073,Z 486.328,A -85,B 0,C 180,E1 -19458.624,E2 -19458.624} C_VEL
LIN {X 0,Y 242.013,Z 486.336,A -85,B 0,C 180,E1 -19462.18,E2 -19462.18} C_VEL
LIN {X 0,Y 242.066,Z 486.33,A -85,B 0,C 180,E1 -19465.838,E2 -19465.838} C_VEL
LIN {X 0,Y 242.006,Z 486.339,A -85,B 0,C 180,E1 -19469.583,E2 -19469.583} C_VEL
LIN {X 0,Y 241.991,Z 486.342,A -85,B 0,C 180,E1 -19473.491,E2 -19473.491} C_VEL
LIN {X 0,Y 242.013,Z 486.337,A -85,B 0,C 180,E1 -19477.577,E2 -19477.577} C_VEL
LIN {X 0,Y 242.138,Z 486.322,A -85,B 0,C 180,E1 -19482.693,E2 -19482.693} C_VEL
LIN {X 0,Y 242.219,Z 486.611,A -85,B 0,C 180,E1 -19483.5,E2 -19483.5} C_VEL
LIN {X 0,Y 243.251,Z 492.38,A -85,B 0,C 180,E1 -19488.693,E2 -19488.693} C_VEL
LIN {X 0,Y 243.765,Z 495.182,A -85,B 0,C 180,E1 -19491.118,E2 -19491.118} C_VEL
LIN {X 0,Y 243.966,Z 498.339,A -85,B 0,C 180,E1 -19493.765,E2 -19493.765} C_VEL
LIN {X 0,Y 243.444,Z 501,A -85,B 0,C 180,E1 -19495.924,E2 -19495.924} C_VEL
LIN {X 0,Y 242.4,Z 502.662,A -85,B 0,C 180,E1 -19497.237,E2 -19497.237} C_VEL
LIN {X 0,Y 238.964,Z 505.392,A -85,B 0,C 180,E1 -19499.354,E2 -19499.354} C_VEL
LIN {X 0,Y 236.121,Z 507.563,A -85,B 0,C 180,E1 -19501.082,E2 -19501.082} C_VEL
LIN {X 0,Y 234.798,Z 509.224,A -85,B 0,C 180,E1 -19502.438,E2 -19502.438} C_VEL
LIN {X 0,Y 234.627,Z 509.787,A -85,B 0,C 180,E1 -19502.901,E2 -19502.901} C_VEL
LIN {X 0,Y 233.965,Z 513.964,A -85,B 0,C 180,E1 -19506.37,E2 -19506.37} C_VEL
LIN {X 0,Y 234.592,Z 526.563,A -85,B 0,C 180,E1 -19507.368,E2 -19507.368} C_VEL
LIN {X 0,Y 235.667,Z 539.647,A -85,B 0,C 180,E1 -19508.721,E2 -19508.721} C_VEL
LIN {X 0,Y 236.942,Z 553.241,A -85,B 0,C 180,E1 -19510.507,E2 -19510.507} C_VEL
LIN {X 0,Y 237.567,Z 559.368,A -85,B 0,C 180,E1 -19511.458,E2 -19511.458} C_VEL
LIN {X 0,Y 236.388,Z 569.906,A -85,B 0,C 180,E1 -19513.372,E2 -19513.372} C_VEL
LIN {X 0,Y 235.253,Z 580.505,A -85,B 0,C 180,E1 -19515.732,E2 -19515.732} C_VEL
LIN {X 0,Y 234.334,Z 589.822,A -85,B 0,C 180,E1 -19518.321,E2 -19518.321} C_VEL
LIN {X 0,Y 233.831,Z 597.43,A -85,B 0,C 180,E1 -19520.922,E2 -19520.922} C_VEL
LIN {X 0,Y 233.573,Z 602.803,A -85,B 0,C 180,E1 -19523.188,E2 -19523.188} C_VEL
LIN {X 0,Y 233.501,Z 607.597,A -85,B 0,C 180,E1 -19525.685,E2 -19525.685} C_VEL
LIN {X 0,Y 233.541,Z 611.385,A -85,B 0,C 180,E1 -19528.276,E2 -19528.276} C_VEL
LIN {X 0,Y 233.608,Z 613.326,A -85,B 0,C 180,E1 -19530,E2 -19530} C_VEL
LIN {X 0,Y 233.316,Z 614.741,A -85,B 0,C 180,E1 -19531.727,E2 -19531.727} C_VEL
LIN {X 0,Y 232.969,Z 616.407,A -85,B 0,C 180,E1 -19535.193,E2 -19535.193} C_VEL
LIN {X 0,Y 233.169,Z 616.581,A -85,B 0,C 180,E1 -19538.668,E2 -19538.668} C_VEL
LIN {X 0,Y 234.179,Z 615.284,A -85,B 0,C 180,E1 -19542.127,E2 -19542.127} C_VEL
LIN {X 0,Y 236.094,Z 612.608,A -85,B 0,C 180,E1 -19545.54,E2 -19545.54} C_VEL
LIN {X 0,Y 239.094,Z 608.52,A -85,B 0,C 180,E1 -19548.865,E2 -19548.865} C_VEL
LIN {X 0,Y 242.079,Z 604.082,A -85,B 0,C 180,E1 -19551.53,E2 -19551.53} C_VEL
LIN {X 0,Y 246.525,Z 597.739,A -85,B 0,C 180,E1 -19554.417,E2 -19554.417} C_VEL
LIN {X 0,Y 251.481,Z 590.39,A -85,B 0,C 180,E1 -19557.009,E2 -19557.009} C_VEL
LIN {X 0,Y 256.929,Z 581.657,A -85,B 0,C 180,E1 -19559.497,E2 -19559.497} C_VEL
LIN {X 0,Y 259.364,Z 576.312,A -85,B 0,C 180,E1 -19560.988,E2 -19560.988} C_VEL
LIN {X 0,Y 261.77,Z 568.362,A -85,B 0,C 180,E1 -19563.414,E2 -19563.414} C_VEL
LIN {X 0,Y 263.228,Z 560.834,A -85,B 0,C 180,E1 -19565.972,E2 -19565.972} C_VEL
LIN {X 0,Y 264.173,Z 554.642,A -85,B 0,C 180,E1 -19568.39,E2 -19568.39} C_VEL
LIN {X 0,Y 264.492,Z 552,A -85,B 0,C 180,E1 -19569.623,E2 -19569.623} C_VEL
LIN {X 0,Y 264.54,Z 548.846,A -85,B 0,C 180,E1 -19571.619,E2 -19571.619} C_VEL
LIN {X 0,Y 264.717,Z 546.058,A -85,B 0,C 180,E1 -19574.207,E2 -19574.207} C_VEL
LIN {X 0,Y 264.821,Z 544.988,A -85,B 0,C 180,E1 -19576.37,E2 -19576.37} C_VEL
LIN {X 0,Y 264.869,Z 545.089,A -85,B 0,C 180,E1 -19578.445,E2 -19578.445} C_VEL
LIN {X 0,Y 265.235,Z 545.793,A -85,B 0,C 180,E1 -19580.511,E2 -19580.511} C_VEL
LIN {X 0,Y 266.04,Z 547.967,A -85,B 0,C 180,E1 -19583.382,E2 -19583.382} C_VEL
LIN {X 0,Y 266.352,Z 550.497,A -85,B 0,C 180,E1 -19585.291,E2 -19585.291} C_VEL
LIN {X 0,Y 266.532,Z 554.303,A -85,B 0,C 180,E1 -19587.543,E2 -19587.543} C_VEL
LIN {X 0,Y 266.246,Z 558.197,A -85,B 0,C 180,E1 -19589.413,E2 -19589.413} C_VEL
LIN {X 0,Y 265.76,Z 559.499,A -85,B 0,C 180,E1 -19589.838,E2 -19589.838} C_VEL
LIN {X 0,Y 259.776,Z 568.596,A -85,B 0,C 180,E1 -19592.181,E2 -19592.181} C_VEL
LIN {X 0,Y 254.341,Z 576.032,A -85,B 0,C 180,E1 -19594.641,E2 -19594.641} C_VEL
LIN {X 0,Y 250.129,Z 581.241,A -85,B 0,C 180,E1 -19596.836,E2 -19596.836} C_VEL
LIN {X 0,Y 245.319,Z 586.635,A -85,B 0,C 180,E1 -19599.893,E2 -19599.893} C_VEL
LIN {X 0,Y 241.395,Z 590.505,A -85,B 0,C 180,E1 -19603.074,E2 -19603.074} C_VEL
LIN {X 0,Y 239.639,Z 591.889,A -85,B 0,C 180,E1 -19604.696,E2 -19604.696} C_VEL
LIN {X 0,Y 237.02,Z 593.542,A -85,B 0,C 180,E1 -19608.021,E2 -19608.021} C_VEL
LIN {X 0,Y 234.914,Z 593.824,A -85,B 0,C 180,E1 -19611.397,E2 -19611.397} C_VEL
LIN {X 0,Y 233.883,Z 592.598,A -85,B 0,C 180,E1 -19614.828,E2 -19614.828} C_VEL
LIN {X 0,Y 233.192,Z 589.91,A -85,B 0,C 180,E1 -19618.273,E2 -19618.273} C_VEL
LIN {X 0,Y 233.023,Z 586.838,A -85,B 0,C 180,E1 -19620.864,E2 -19620.864} C_VEL
LIN {X 0,Y 233.082,Z 582.801,A -85,B 0,C 180,E1 -19623.458,E2 -19623.458} C_VEL
LIN {X 0,Y 233.28,Z 577.428,A -85,B 0,C 180,E1 -19626.175,E2 -19626.175} C_VEL
LIN {X 0,Y 233.733,Z 571.397,A -85,B 0,C 180,E1 -19628.647,E2 -19628.647} C_VEL
LIN {X 0,Y 234.407,Z 563.651,A -85,B 0,C 180,E1 -19631.238,E2 -19631.238} C_VEL
LIN {X 0,Y 235.372,Z 554.123,A -85,B 0,C 180,E1 -19633.821,E2 -19633.821} C_VEL
LIN {X 0,Y 236.65,Z 543.559,A -85,B 0,C 180,E1 -19636.166,E2 -19636.166} C_VEL
LIN {X 0,Y 238.013,Z 531.725,A -85,B 0,C 180,E1 -19638.285,E2 -19638.285} C_VEL
LIN {X 0,Y 239.147,Z 520.434,A -85,B 0,C 180,E1 -19639.937,E2 -19639.937} C_VEL
LIN {X 0,Y 237.277,Z 509.333,A -85,B 0,C 180,E1 -19641.327,E2 -19641.327} C_VEL
LIN {X 0,Y 234.611,Z 494.497,A -85,B 0,C 180,E1 -19642.824,E2 -19642.824} C_VEL
LIN {X 0,Y 233.542,Z 487.397,A -85,B 0,C 180,E1 -19643.441,E2 -19643.441} C_VEL
LIN {X 0,Y 233.854,Z 487.357,A -85,B 0,C 180,E1 -19646.795,E2 -19646.795} C_VEL
LIN {X 0,Y 234.259,Z 487.303,A -85,B 0,C 180,E1 -19650.666,E2 -19650.666} C_VEL
